# B&R Automation Studio project TD52 (part 7)

#### GeACtr.st
```iecst
(********************************************************************
 * COPYRIGHT -- INNIO Company
 ********************************************************************
 * Package:
 * File: GeACtr.st
 * Author: maierm
 * Created: May 22, 2012
 *******************************************************************)

(* ******************************************************************
 * History:
 *
 * V0.10.0		22-05-2012 maierm, 	generated
 * V0.10.1		21-06-2012 maierm, 	set clamp at line 102
 *								  	tProcPar.valid commented
 *								   	line 321 simplified - if / else
 *									was not necessary
 * V0.20.0		22-04-2013 maierm,	Datatype tParameter.Kp_manualAdjust, tParameter.Tn_manualAdjust and tParameter.Tv_manualAdjust
 *									changed to REAL, scaling included:
 *										tInput.Y_man 				==> tInput.Y_man * SCALE_PERCENT
 *										tInput.Y_set 				==> tInput.Y_set * SCALE_PERCENT
 *										tInput.A	 				==> tInput.A * SCALE_PERCENT
 *										tOutput.Y	 				==> rY / SCALE_PERCENT
 *										tOutput.e	 				==> xLCRPID.e / SCALE_PERCENT
 *										tOutput.Tn_tune 			==> tProcPar.Tn_tune * SCALE_TIME
 *										tOutput.Tv_tune 			==> tProcPar.Tv_tune * SCALE_TIME
 *										tParameter.Y_min   			==> tParameter.Y_min * SCALE_PERCENT
 *										tParameter.Y_max   			==> tParameter.Y_max * SCALE_PERCENT
 *										tParameter.dY_max  			==> tParameter.dY_max * SCALE_PERCENT
 *										tParameter.Y_block 			==> tParameter.Y_block * SCALE_PERCENT
 *										tParameter.Tn	   			==> tParameter.Tn / SCALE_TIME
 *										tParameter.Tv	   			==> tParameter.Tv / SCALE_TIME
 *										tParameter.Kp_manualAdjust 	==> tParameter.Kp_manualAdjust * SCALE_PERCENT
 *										tParameter.Tn_manualAdjust  ==> tParameter.Tn_manualAdjust * SCALE_PERCENT
 *										tParameter.Tv_manualAdjust 	==> tParameter.Tv_manualAdjust * SCALE_PERCENT
 *										tParameter.t_min_pulse_up 	==> tParameter.t_min_pulse_up / SCALE_TIME
 *										tParameter.t_period_up 		==> tParameter.t_period_up / SCALE_TIME
 *										tParameter.t_min_pulse_down ==> tParameter.t_min_pulse_down / SCALE_TIME
 *										tParameter.t_period_down 	==> tParameter.t_period_down / SCALE_TIME
 * V0.30.0		11-06-2013 maierm, 	comment format changed,
 *								   	corrected bug in part "input pwm up" and "input pwm down" -
 *								   	instead of bSafe2 was bSafe1 written - correct is bSafe2,
 *								   	changed rYmin to tParameter.Y_min in part "reset tuning or pid error",
 *								   	changed rYmax to tParameter.Y_max in part "reset tuning or pid error",
 *								   	set X to W for one cycle at enable of the fub
 * V0.40.0		27-06-2013 maierm, 	status of LCRPWM_up and LCRPWM_down has the lowest priority,
 *								   	instead of manuel mode, Input.Y_man is always following Output.Y,
 *								   	setting the internal I - component of the LCRPIDTune FUB directly to the new Y_min and Y_max limits
 * V0.50.0		28.06.2013 maierm, 	tInput.enable = FALSE sets the LCRPID to manual mode. LCRPID and LCRPIDTune is always running
 * V0.60.0		03.07.2013 Tinello,	Change tOutput.e  ==> Difference between W and X
 * V0.60.1		03.09.2013 maierm, 	bug at the feature "setting the internal I - component of the LCRPIDTune..." removed (Comparison
 *								   	between scaled and not scaled value)
 * V0.60.2		02.12.2013 Tinello,	If Y_Min = Y_Max -> automatic adjustment of Y_Min and Y_Max
 *									automatic limitation of Y_Min and Y_Max to -100% to 100%
 * V0.60.3		24.09.2016 Fahring,	set tAddPar.Kfbk = 1.0 to activate anti wind up protection
									set tAddPar.Tf_Tv = 0.1 / default value
 * V0.60.4		11.01.2017 Tinello,	Setpoint ramp changed from stage per second to linear ramp according to used cycle time
 * V0.70.0		25.01.2022 Perktold,Parameters: added W_set2, and GeinScheduling PID values; deleted "_manualAdjust" Parameters
									added Inputs: 	W_set2_Active, Retrigger, GainScheduling, Y_min_cust, Y_max_cust, AlwaysUseYRamp, KeepYManAtBlock
									added Outputs: 	Y_min_act, Y_max_act, Kp_act, Tn_act, Tv_act, Yp, Yi, Yd, BlockAutoTune, Show_PID_act
									LCRPWM replaced by LCRContinServo for sept_up/down output computation
 ****************************************************************************************************************************************************)

FUNCTION_BLOCK GeACtr

	(* ******************************** *)
	(*				ACCESS				*)
	(* ******************************** *)

	tParameter ACCESS pParameter; 								(* parameter from user *)
	tInput 	   ACCESS pInput;	  								(* input from user *)
	tOutput    ACCESS pOutput;	 								(* output from user *)
	tProcPar   ACCESS ADR(xLCRPIDTune.processPar);				(* Kp, Tn, Tv from LCRPIDTune *)

	(* ************************************************ *)
	(*	enable / auto / man / safe1 / safe2 / Retrigger	*)
	(* ************************************************ *)

	xR_TRIG_enable(CLK := tInput.enable);						(* generate rising trigger at enable*)
	bAuto  := tInput.enable AND NOT(tInput.Y_man_Active);		(* automatic *)
	bMan   := tInput.enable AND tInput.Y_man_Active;			(* manual *)
	bSafe1 := NOT(tInput.enable) AND NOT(tInput.Y_set_Active);	(* 1st safe - Y_block *)
	bSafe2 := NOT(tInput.enable) AND tInput.Y_set_Active;		(* 2nd safe - Y_set *)
	xR_TRIG_Retrigger(CLK := tInput.Retrigger);					(* generate rising trigger at retrigger*)

	(* ******************************** *)
	(*				  W					*)
	(* ******************************** *)

	tParameter.W_set := LIMIT(tParameter.W_min, tParameter.W_set, tParameter.W_max);	(* limit W from visu *)
	tParameter.W_set2 := LIMIT(tParameter.W_min, tParameter.W_set2, tParameter.W_max);	(* limit W from visu *)

	IF tInput.W_ext_Active 	THEN rWSet := tInput.W_ext; 					(* W from external *)
						 	ELSE
								IF tInput.W_set2_Active THEN
									rWSet := tParameter.W_set2;				(* W from visu - second internal set point*)
								ELSE
									rWSet := tParameter.W_set;				(* W from visu *)
								END_IF
							END_IF

	xLCRRamp_WSet.enable 	:= TRUE;
	xLCRRamp_WSet.dy_up 	:= tParameter.dW_up;							(* ramp up:   value/s *)
	xLCRRamp_WSet.dy_down 	:= tParameter.dW_down;							(* ramp down: value/s *)
	xLCRRamp_WSet.y_min 	:= tParameter.W_min;							(* limit W actual *)
	xLCRRamp_WSet.y_max 	:= tParameter.W_max;							(* limit W actual *)
	xLCRRamp_WSet.y_set 	:= tInput.X;									(* set X to W at enable of fub or retriggering *)
	xLCRRamp_WSet.set 		:= xR_TRIG_enable.Q OR xR_TRIG_Retrigger.Q;		(* activate set in case of retriggering or at enable of fub *)
	xLCRRamp_WSet(x 		:= rWSet);

	rW := LIMIT(tParameter.W_min, xLCRRamp_WSet.y, tParameter.W_max);		(* limit W *)
	tOutput.W 	:= rW; 														(* W actual *)

	(* ******************************** *)
	(*	 Y_min / Y_max (error 12037)	*)
	(* ******************************** *)

	IF (tParameter.Y_min <> rYMinOld) AND (tParameter.Y_min > tParameter.Y_max) THEN		(* Limit Y_min parameter to Y_max if Y_min > Y_max*)
		tParameter.Y_min := tParameter.Y_max;
	END_IF
	IF (tParameter.Y_max <> rYMaxOld) AND (tParameter.Y_max < tParameter.Y_min) THEN		(* Limit Y_max parameter to Y_min if Y_max < Y_min*)
		tParameter.Y_max := tParameter.Y_min;
	END_IF

	IF (tParameter.Y_max > Y_MAX  			OR												(* create error 12037 manually because of a bug in V2.80.1 *)
		tParameter.Y_min < Y_MIN 			OR
		tParameter.Y_max < tParameter.Y_min)
	THEN
		rYMax := 0;	 																		(* set Ymax to 0 *)
		rYMin := 0;  																		(* set Ymin to 0 *)
	ELSE
		rYMax := LIMIT(-1.0, MAX(MIN(tParameter.Y_max, tInput.Y_max_cust), MAX(tParameter.Y_min, tInput.Y_min_cust)), 1.0) * SCALE_PERCENT;	(* include Y_min_cust & Y_max_cust *)
		rYMin := LIMIT(-1.0, MIN(MAX(tParameter.Y_min, tInput.Y_min_cust), MIN(tParameter.Y_max, tInput.Y_max_cust)), 1.0) * SCALE_PERCENT;	(* include Y_min_cust & Y_max_cust *)
	END_IF

	IF rYMax = rYMin THEN																	(* in case Ymax = Ymin set them 0.01 appart *)
		IF rYMax >= 0 THEN	rYMin := rYMax - 0.01; 	END_IF
		IF rYMax < 0 THEN	rYMax := rYMin + 0.01; 	END_IF
	END_IF

	(* put the resulting YMin & YMax to the output structure *)
	tOutput.Y_max_act	:=	rYMax / SCALE_PERCENT;
	tOutput.Y_min_act	:=	rYMin / SCALE_PERCENT;

	(* If Y_min or Y_max is changed, the internal I - component of the LCRPIDTune FUB ran through the whole range to the new Y_min and
	(* Y_max limits. This behavior is optimised by setting the internal I - component of the LCRPIDTune FUB directly to the new Y_min and
	(* Y_max limits *)
	IF (rYMin <> rYMinintOld OR rYMax <> rYMaxintOld) THEN
		pYi1 ACCESS ADR(xLCRPIDTune.internal_data.Yi1); 									(* internal I - component can't be changed directly *)

		IF 	  (tOutput.Y <= (rYMin / SCALE_PERCENT)) THEN	pYi1 := rYMin;					(* set the internal I - component directly *)
		ELSIF (tOutput.Y >= (rYMax / SCALE_PERCENT)) THEN	pYi1 := rYMax;	END_IF			(* set the internal I - component directly *)
	END_IF

	IF xR_TRIG_Retrigger.Q OR xR_TRIG_enable.Q THEN											(* in case of retriggering or at enable of fub     *)
		pYi1 ACCESS ADR(xLCRPIDTune.internal_data.Yi1); 									(* access the internal integrator value of the CTR *)
		pYi1 := tOutput.Y * SCALE_PERCENT;													(* set the integrator to represent the last Y      *)
	END_IF;

	(* ******************************** *)
	(*				Tuning				*)
	(* ******************************** *)

	(* limit gain scheduling input from 0 to 1*)
	tInput.GainScheduling	:= LIMIT(0.0, tInput.GainScheduling, 1.0);

	(* Generate Output for VISU to decide if Parameters or actual PID-values are shown *)
	IF (tInput.GainScheduling >= 0.01) THEN
		tOutput.Show_PID_act	:= TRUE;		(* not show PID-paramters - show actual PID-values instead *)
	ELSE
		tOutput.Show_PID_act	:= FALSE;		(* show PID-paramters *)
	END_IF;

	(* De-/Activation of the Auto Tune function *)
	IF 	(xLCRPIDTune.status = 65534) 	OR		(* Auto Tune inactive (eg. Controller not enabled) *)
		(tInput.GainScheduling >= 0.01)	OR 		(* Gain Scheduling active - don't show parameters - show actual values instead *)
		NOT tInput.enable				OR		(* Controller nor enabled *)
		bMan									(* Controller running in manual mode *)
	THEN
		tInput.Tune_start 		:= FALSE;		(* reset *)
		tOutput.BlockAutoTune	:= TRUE;		(* lock VISU Button for AUTO Tune *)
	ELSE
		tOutput.BlockAutoTune	:= FALSE;		(* unlock VISU Button for AUTO Tune *)
	END_IF;

	(* tuning enable *)
	bTune_enable := TRUE;

	(* start *)
	IF (tInput.Tune_start = TRUE AND bAuto = TRUE AND usTune_status = 0) THEN (* user start *)
		bTune_active        := TRUE; 					(* tuning started *)
		bTunePIOld			:= tInput.Tune_PI;  		(* store *)
		bTunePIDOld			:= tInput.Tune_PID; 		(* store *)
		xLCRPIDTune.request := xTunReq(tInput.Tune_PI, tInput.Tune_PID, tInput.Tune_quality, tParameter.invert); (* calculate tuning request *)
	END_IF
	tInput.Tune_start 		:= FALSE;	(* reset *)

	(* stop *)
	IF (tInput.Tune_stop = TRUE 										OR 		(* user stop *)
		EDGENEG(bAuto) = TRUE											OR  	(* fub enable = FALSE OR manual = TRUE *)
		tAddPar.invert <> tParameter.invert 							OR  	(* invert parameter changed *)
		(xLCRPIDTune.status >= 12025 AND xLCRPIDTune.status <> 65534)) 			(* error happened *)
	THEN
		xLCRPIDTune.request := LCRPID_TUNE_REQU_OFF; 							(* deactivate tuning *)
		usTune_status       := 0; 												(* reset *)
		bTune_save 		    := FALSE; 											(* tuning stopped *)
		bTune_active        := FALSE; 											(* tuning stopped *)

		IF (xLCRPIDTune.status >= 12025 AND xLCRPIDTune.status <> 65534) THEN	(* tuning error *)
			usTune_status := xLCRPIDTune.status;								(* error status *)
			IF (xLCRPIDTune.status = 12039)	THEN
				usTune_status := xLCRPIDTune.addInfo;							(* show additional info *)
			ELSIF (xLCRPIDTune.status = 31564) THEN
				xResErr(ADR(bTune_enable), xLCRPIDTune.status);					(* reset enable after error *)
			END_IF
		END_IF
	END_IF
	tInput.Tune_stop := FALSE;			(* reset *)

	(* store tuning parameter *)
	IF (tInput.Tune_takeover = TRUE) THEN 						(* get tuning parameter every time *)
		bTune_save 	  		:= FALSE; 							(* tuning save closed *)
		usTune_status 		:= 0;	    						(* set status - no error / tuning finished / parameter saved *)
		tParameter.Kp 		:= tOutput.Kp_tune;
		tParameter.Tn 		:= tOutput.Tn_tune;
		tParameter.Tv 		:= tOutput.Tv_tune;
	END_IF
	tInput.Tune_takeover	:= FALSE; 	(* reset *)

	(* set ctrl parameter *)
	IF (bTune_active = FALSE AND bTune_save = TRUE) THEN 		(* no tuning / tuning parameter not set *)
		IF (bTunePIOld = TRUE AND bTunePIDOld = FALSE) THEN 	(* PI - tuning *)
			tProcPar.Tv_tune := 0;		(* delete D *)
		ELSIF (bTunePIOld = FALSE AND bTunePIDOld = FALSE) THEN (* P - tuning *)
			tProcPar.Tn_tune := 0;		(* delete I *)
			tProcPar.Tv_tune := 0;		(* delete D *)
		END_IF
		tOutput.Kp_tune := tProcPar.Kp_tune; 			  		(* fub to tune parameter *)
		tOutput.Tn_tune := tProcPar.Tn_tune * SCALE_TIME; 		(* fub to tune parameter *)
		tOutput.Tv_tune := tProcPar.Tv_tune * SCALE_TIME; 		(* fub to tune parameter *)

	ELSIF (bTune_active = FALSE AND bTune_save = FALSE) THEN 	(* no tuning and parameter set *)
		tProcPar.valid   := TRUE; 										(* necessary for the LCRPIDTune(). Kp_tune, Tn_tune and Tv_tune *)
																		(* are "valid" and can be used from the FUB 					*)
		(* Interpolate PID-Parameters via Gain Scheduling *)
		tProcPar.Kp_tune :=  (1.0 - tInput.GainScheduling) * tParameter.Kp + tInput.GainScheduling * tParameter.Kp_GainScheduling; 						(* parameter to fub *)
		tProcPar.Tn_tune := ((1.0 - tInput.GainScheduling) * tParameter.Tn + tInput.GainScheduling * tParameter.Tn_GainScheduling) / SCALE_TIME; 		(* parameter to fub *)
		tProcPar.Tv_tune := ((1.0 - tInput.GainScheduling) * tParameter.Tv + tInput.GainScheduling * tParameter.Tv_GainScheduling) / SCALE_TIME; 	 	(* parameter to fub *)
		IF xR_TRIG_Retrigger.Q OR xR_TRIG_enable.Q THEN
			tProcPar.Tv_tune := 0;
		END_IF;
	END_IF

	(* tuning status *)
	IF (bTune_active = FALSE AND bTune_save = TRUE) THEN
		usTune_status := 1; 									(* set status - tuning finished, but not closed *)
	ELSIF (bTune_active = TRUE) THEN
		usTune_status := 2;										(* set status - tuning active *)
	END_IF

	(* parameter *)
	xLCRPIDTune.enable 			:= bTune_enable;
	xLCRPIDTune.Y_min  			:= rYMin;
	xLCRPIDTune.Y_max  			:= rYMax;
	xLCRPIDTune.X_min  			:= tInput.X_min;
	xLCRPIDTune.X_max  			:= tInput.X_max;
	xLCRPIDTune.P_manualAdjust 	:= 0;
	xLCRPIDTune.I_manualAdjust 	:= 0;
	xLCRPIDTune.D_manualAdjust 	:= 0;

	(* additional parameter *)
	tAddPar.dY_max      		:= tParameter.dY_max * SCALE_PERCENT;
	tAddPar.deadband    		:= tParameter.deadband;
	tAddPar.d_mode      		:= LCRPID_D_MODE_E;
	tAddPar.invert	    		:= tParameter.invert;
	tAddPar.Kfbk				:= 1.0;
	tAddPar.Tf_Tv				:= 0.1;
	xLCRPIDTune.pAddPar 		:= ADR(tAddPar);	 (* additional parameter *)

	(* reset valid *)
	IF (EDGEPOS(bTune_active) = TRUE) THEN 	(* new tuning *)
		tProcPar.valid 			:= FALSE;  	(* reset necessary at new tuning - otherwise ctrl fub is immediately finished *)
	END_IF

	xLCRPIDTune();

	(* put the resulting PID-values to the output structure *)
	tOutput.Kp_act	:= tProcPar.Kp_tune;
	tOutput.Tn_act	:= tProcPar.Tn_tune * SCALE_TIME;
	tOutput.Tv_act	:= tProcPar.Tv_tune * SCALE_TIME;

	(* store during tuning the parameters from the visu to the internal structure (if user changed it during the tuning) *)
	IF (bTune_active = TRUE AND xLCRPIDTune.state < LCRPID_TUNE_STATE_RESET_CNTL) THEN
		tProcPar.Kp_tune 	  := tParameter.Kp; 			 (* parameter to fub *)
		tProcPar.Tn_tune 	  := tParameter.Tn / SCALE_TIME; (* parameter to fub *)
		tProcPar.Tv_tune 	  := tParameter.Tv / SCALE_TIME; (* parameter to fub *)
	END_IF

	(* set parameter after enable = TRUE (LCRPID sets parameter to 0 / 0.5 aso. after enable = TRUE) *)
	IF (EDGEPOS(tInput.enable) = TRUE) THEN
		tProcPar.valid   	  := TRUE; 		   				 (* valid necessary that controller use the parameters - after enable = TRUE *)
		tProcPar.Kp_tune 	  := tParameter.Kp; 			 (* parameter to fub *)
		tProcPar.Tn_tune 	  := tParameter.Tn / SCALE_TIME; (* parameter to fub *)
		tProcPar.Tv_tune 	  := tParameter.Tv / SCALE_TIME; (* parameter to fub *)
	END_IF

	(* tuning finished *)
	IF (bTune_active = TRUE AND xLCRPIDTune.state = LCRPID_TUNE_STATE_FINISHED) THEN
		xLCRPIDTune.request   := LCRPID_TUNE_REQU_OFF; 		(* deactivate tuning *)
		bTune_save 		      := TRUE;  					(* save parameter *)
		bTune_active          := FALSE; 					(* tuning finished *)

		(* error 12041 manually *)
		IF (tProcPar.valid = FALSE AND rW <> rWOld) THEN	(* set status 12041 manually because of a bug in V2.80.1 *)
			rWOld 		      := rW;
			bTune_save        := FALSE;
			usTune_status     := 12041;
		END_IF
	END_IF

	(* error 12041 manually *)
	IF (bTune_active = FALSE) THEN
		rWOld := rW;
	END_IF

	(* ******************************** *)
	(*				PID					*)
	(* ******************************** *)

	(* error *)
	IF (xLCRPID.status >= 12025 AND xLCRPID.status <> 65534) THEN	 (* error happened *)
		usPID_status := xLCRPID.status;	 			(* show error number *)
	ELSE
		usPID_status := 0;
	END_IF

	(* Y manual *)
	IF (bSafe1 = TRUE) THEN											(* first safe value *)
		IF tInput.KeepYManAtBlock THEN								(* prevent overriding of tInput.Y_man *)
			xLCRPID.Y_man:= tParameter.Y_block * SCALE_PERCENT;		(* write Y_block value to LCRPID directly *)
		ELSE
			tInput.Y_man := tParameter.Y_block;						(* override Y_man with Y_block value*)
		END_IF;
		xLCRPID.mode := LCRPID_MODE_MAN_JOLTFREE;					(* PID manual mode *)
	END_IF

	IF (bSafe2 = TRUE) THEN 										(* second safe value *)
		IF tInput.KeepYManAtBlock THEN								(* prevent overriding of tInput.Y_man *)
			xLCRPID.Y_man:= tInput.Y_set * SCALE_PERCENT;			(* write Y_set value to LCRPID directly *)
		ELSE
			tInput.Y_man := tInput.Y_set;							(* override Y_man with Y_set value*)
		END_IF
		xLCRPID.mode := LCRPID_MODE_MAN_JOLTFREE;					(* PID manual mode *)
	END_IF

	IF (bAuto = TRUE) THEN											(* automatic mode *)
		tInput.Y_man := tOutput.Y;									(* in automatic mode Y_man is following Y *)
		xLCRPID.Y_man:= tInput.Y_man * SCALE_PERCENT;				(* write Y_man value to LCRPID directly *)
		xLCRPID.mode := LCRPID_MODE_AUTO;							(* PID automatic mode *)
	END_IF

	IF (bMan = TRUE) THEN																	(* manual mode *)
		tInput.Y_man := LIMIT(rYMin / SCALE_PERCENT, tInput.Y_man, rYMax / SCALE_PERCENT);	(* limit Y manual from visu *)
		xLCRPID.Y_man := tInput.Y_man * SCALE_PERCENT;										//Y_man for LCRPID acc Y_man
		xLCRPID.mode := LCRPID_MODE_MAN_JOLTFREE;											(* PID manual mode *)
	END_IF

	IF NOT tInput.KeepYManAtBlock THEN
		xLCRPID.Y_man 	 := tInput.Y_man * SCALE_PERCENT;									(* transfer Y_man value to LCRPID *)
	END_IF;

	(* parameter *)
	xLCRPID.enable 	 := TRUE;
	xLCRPID.ident  	 := xLCRPIDTune.ident;
	xLCRPID.Y_max  	 := rYMax;
	xLCRPID.Y_min  	 := rYMin;
	xLCRPID.A	   	 := tInput.A * SCALE_PERCENT;
	xLCRPID.W 		 := rW;		   					(* W *)
	xLCRPID.X 		 := tInput.X;  					(* X *)
	xLCRPID();

	rY 		  		 := xLCRPID.Y;					(* Y FuB *)
	tOutput.e 		 := xLCRPID.X - xLCRPID.W;		(* Error = X - W *)

	(* ******************************** *)
	(*				  Y 				*)
	(* ******************************** *)

	(* change of request *)
	IF ((EDGEPOS(bTune_active) = TRUE) OR 							(* set Y to Y old after start of tuning *)
		(EDGENEG(bTune_active) = TRUE AND bTune_save = FALSE)) 		(* set Y to Y old after tuning stop 	*)
	THEN
		rY := rYOld;	(* Y decreases minimal for one cycle after start of tuning and cancel of tuning	*)
					   	(* - set Y to YOld for one cycle compensate this decrease 						*)
	END_IF
	rYOld := rY;

	(* first safe value *)
	IF (bSafe1 = TRUE) THEN
		rY := tParameter.Y_block * SCALE_PERCENT;	(* Y_block *)
	END_IF

	(* second safe value *)
	IF (bSafe2 = TRUE) THEN
		rY := tInput.Y_set * SCALE_PERCENT;			(* Y_set *)
	END_IF

	(* additional ramp at the end of the controller to prohibit step changes on Y *)
	xLCRRamp_Y.enable 	:= TRUE;
	xLCRRamp_Y.dy_up 	:= tParameter.dY_max;			(* ramp up:   value/s *)
	xLCRRamp_Y.dy_down 	:= tParameter.dY_max;			(* ramp down: value/s *)
	xLCRRamp_Y.y_min 	:= -1.0;						(* limit Y actual - full range *)
	xLCRRamp_Y.y_max 	:=  1.0;						(* limit Y actual - full range *)
	xLCRRamp_Y.y_set 	:= rY / SCALE_PERCENT;
	xLCRRamp_Y.set 		:= NOT tInput.AlwaysUseYRamp;	(* possibility to deactivate the ramp *)
	xLCRRamp_Y(x 		:= (rY / SCALE_PERCENT));

	tOutput.Y := xLCRRamp_Y.y; 				(* Y to output *)

	(* transfer all parts of Y to the tOutput structure *)
	tOutput.Yp		:= xLCRPID.Yp / SCALE_PERCENT;
	tOutput.Yi		:= xLCRPID.Yi / SCALE_PERCENT;
	tOutput.Yd		:= xLCRPID.Yd / SCALE_PERCENT;

	(* ******************************** *)
	(*				PWM					*)
	(* ******************************** *)
	IF tInput.StepperMode THEN
		(* PWM Up *)
		(* enable *)
		bPWM_up_enable := tInput.enable;		(* activate *)
		xResChg(ADR(bPWM_up_enable), tParameter.t_min_pulse_up / SCALE_TIME, xLCRPWM_up.t_min_pulse);		(* reset enable if t_min_pulse
																											   changed *)
		(* parameter *)
		xLCRPWM_up.enable 	   := bPWM_up_enable;
		xLCRPWM_up.max_value   := rYMax;
		xLCRPWM_up.min_value   := xCalMid(rYMin, rYMax);		(* calculate middle of Y_max / Y_min range *)
		xLCRPWM_up.t_min_pulse := tParameter.t_min_pulse_up / SCALE_TIME;
		xLCRPWM_up.t_period	   := tParameter.t_period_up / SCALE_TIME;

		(* input PWM Up *)
		IF (bSafe1 = TRUE OR bSafe2 = TRUE OR bMan = TRUE) 		(* Y_block / Y_set / Y_man *)
		THEN
			xLCRPWM_up.x := xCalMid(rYMin, rYMax); 				(* restrict input to middle of Y_max / Y_min range *)
		ELSE
			xLCRPWM_up.x := rY; 								(* actual value *)
		END_IF

		xLCRPWM_up();

		(* PWM Down *)
		(* enable *)
		bPWM_down_enable := tInput.enable;		(* activate *)
		xResChg(ADR(bPWM_down_enable), tParameter.t_min_pulse_down / SCALE_TIME, xLCRPWM_down.t_min_pulse);	(* reset enable if t_min_pulse
																											   changed *)
		(* parameter *)
		xLCRPWM_down.enable 	 := bPWM_down_enable;
		xLCRPWM_down.max_value   := xCalMid(rYMin, rYMax);		(* calculate middle of Y_max / Y_min range *)
		xLCRPWM_down.min_value   := rYMin;
		xLCRPWM_down.t_min_pulse := tParameter.t_min_pulse_down / SCALE_TIME;
		xLCRPWM_down.t_period	 := tParameter.t_period_down / SCALE_TIME;

		(* input PWM Down *)
		IF (bSafe1 = TRUE OR bSafe2 = TRUE OR bMan = TRUE) 		(* Y_block / Y_set / Y_man *)
		THEN
			xLCRPWM_down.x := xCalMid(rYMin, rYMax); 			(* restrict input to middle of Y_max / Y_min range *)
		ELSE
			xLCRPWM_down.x := rY;								(* actual value *)
		END_IF

		xLCRPWM_down();

		(* PWM Up / PWM Down *)
		(* common status for PWM Up and PWM Down *)
		IF 	  (xLCRPWM_up.status   >= 12025) THEN	usPWM_status := xLCRPWM_up.status;
		ELSIF (xLCRPWM_down.status >= 12025) THEN	usPWM_status := xLCRPWM_down.status;
											 ELSE	usPWM_status := 0;				 		END_IF

		(* output only if PWM Up and PWM Down has no error *)
		IF (usPWM_status = 0) THEN
			tOutput.Step_up   := xLCRPWM_up.pulse;
			tOutput.Step_down := NOT(xLCRPWM_down.pulse); 	(* invert necessary *)
		ELSE
			tOutput.Step_up   := FALSE;
			tOutput.Step_down := FALSE;
		END_IF

	ELSE  // tInput.StepperMode = FALSE

		(* ******************************** *)
		(*     continuous servo drive   	*)
		(* ******************************** *)

		(* Enable servo drive *)
		xLCRContinServo.enable        := tInput.enable;

		(* Parameters for continuous servo drive *)
		xLCRContinServo.max_value     := tOutput.Y_max_act;
		xLCRContinServo.min_value     := tOutput.Y_min_act;
		xLCRContinServo.t_impulse     := (tParameter.t_min_pulse_up / 1000) ;
		IF tParameter.dY_max <> 0 THEN
			xLCRContinServo.t_change_up   := (1 / tParameter.dY_max) * (tOutput.Y_max_act - tOutput.Y_min_act);
			xLCRContinServo.t_change_down := (1 / tParameter.dY_max) * (tOutput.Y_max_act - tOutput.Y_min_act);
		END_IF;

		(* Continuous servo drive *)
		xLCRContinServo.x   := tOutput.Y;
		xLCRContinServo();										(* LCRContinServo function block call *)

		(* Copy up and down to controller output *)
		tOutput.Step_up 		:= xLCRContinServo.up;
		tOutput.Step_down 		:= xLCRContinServo.down;
	END_IF;

	(* ******************************** *)
	(*		reset status LCRPIDTune		*)
	(* ******************************** *)

	(* reset tuning or pid error *)
	IF (tParameter.Kp   			<> rKpOld  				OR
		tParameter.Tn 	 			<> rTnOld  				OR
		tParameter.Tv   			<> rTvOld  				OR
		tParameter.Y_min 			<> rYMinOld 			OR
		tParameter.Y_max 			<> rYMaxOld 			OR
		rYMinintOld					<> rYMin				OR
		rYMaxintOld					<> rYMax				OR
		tInput.X_min     			<> rXMinOld 			OR
		tInput.X_max     			<> rXMaxOld 			OR
		tParameter.deadband 		<> rDeadbandOld			OR
		tParameter.dY_max			<> rDYMaxOld)
	THEN
		IF (usTune_status >= 12025 AND usTune_status <> 65534) THEN
			usTune_status := 0;	(* reset tune status after error *)
		END_IF
	END_IF

	rKpOld   			:= tParameter.Kp; (* restore *)
	rTnOld   			:= tParameter.Tn;
	rTvOld   			:= tParameter.Tv;
	rYMinOld 			:= tParameter.Y_min;
	rYMaxOld 			:= tParameter.Y_max;
	rYMinintOld			:= rYMin;
	rYMaxintOld			:= rYMax;
	rXMinOld 			:= tInput.X_min;
	rXMaxOld 			:= tInput.X_max;
	rDeadbandOld      	:= tParameter.deadband;
	rDYMaxOld		  	:= tParameter.dY_max;

	(* ******************************** *)
	(*				Status				*)
	(* ******************************** *)

	tOutput.Active := tInput.enable;

	IF (tInput.enable = TRUE) THEN	(* fub enable *)

		IF 	  (xChkStat(usPID_status)  = TRUE) THEN	tOutput.status := usPID_status;		(* LCRPID state *)
		ELSIF (xChkStat(usTune_status) = TRUE) THEN tOutput.status := usTune_status;	(* LCRTune state *)
		ELSIF (xChkStat(usPWM_status)  = TRUE) THEN tOutput.status := usPWM_status; 	(* LCRPWM_up AND LCRPWM_down state *)
											   ELSE tOutput.status := 0;
		END_IF

	ELSE							(* fub disable *)
		usTune_status  := 0;		(* reset *)
		usPID_status   := 0;
		usPWM_status   := 0;
		bTune_active   := FALSE;
		bTune_save     := FALSE;
		tOutput.status := 65534;	(* status enable = FALSE *)
	END_IF

END_FUNCTION_BLOCK
```

#### GeACtrFunc.st - Functions of the library
```iecst
(********************************************************************
 * COPYRIGHT -- INNIO Company
 ********************************************************************
 * Package:
 * File: GeACtrFunc.st
 * Author: maierm
 * Created: May 22, 2012
 *******************************************************************)

(* ******************************************************************
 * History:
 *
 * V0.1.0		22-05-2012	maierm, generated
 *
 *
 *
 *******************************************************************)

(* returns the middle of min and max value *)
FUNCTION xCalMid

	xCalMid := rMin + (rMax - rMin) / 2;

END_FUNCTION

(* returns TRUE if status is between 0 and 65534  *)
FUNCTION xChkStat

	IF (usActStatus <> 0 AND usActStatus <> 65534) THEN
		xChkStat := TRUE;
	ELSE
		xChkStat := FALSE;
	END_IF

END_FUNCTION

(* switch off the enable if parameter changed *)
FUNCTION xResChg

	bEnable ACCESS pEnable;

	IF (rAct <> rOld) THEN	(* check if old value is different to actual value *)
		bEnable := FALSE;	(* reset *)
	END_IF

	xResChg;

END_FUNCTION

(* reset the enable if an error happened *)
FUNCTION xResErr

	bEnable ACCESS pEnable;

	IF (usStatus >= 12025 AND usStatus <> 65534) THEN	(* switch off enable *)
		bEnable := FALSE;
	END_IF

	xResErr;

END_FUNCTION

(* returns the tuning request *)
FUNCTION xTunReq

	xTunReq := 0;
	xTunReq := xTunReq + LCRPID_TUNE_REQU_OSCILLATE;	(* oscillation *)

	IF (bInvert = TRUE) THEN
		xTunReq := xTunReq + LCRPID_TUNE_REQU_DIR_NEG;		(* negative direction *)
	ELSE
		xTunReq := xTunReq + LCRPID_TUNE_REQU_DIR_POS;		(* positive direction *)
	END_IF

	IF (bPI = TRUE) THEN
		IF (bPID = TRUE) THEN	(* PID tuning *)
			xTunReq := xTunReq + LCRPID_TUNE_REQU_PID;
		ELSE					(* PI tuning *)
			xTunReq := xTunReq + LCRPID_TUNE_REQU_PI;
		END_IF
	ELSE						(* P tuning *)
		xTunReq := xTunReq + LCRPID_TUNE_REQU_P;
	END_IF

	IF (ssQuality = 0) THEN		(* 1 try - 3 periods *)
		xTunReq := xTunReq + LCRPID_TUNE_REQU_OSC_1 + LCRPID_TUNE_REQU_PER_3;
	ELSIF (ssQuality = 1) THEN	(* 2 tries - 4 periods *)
		xTunReq := xTunReq + LCRPID_TUNE_REQU_OSC_2 + LCRPID_TUNE_REQU_PER_4;
	ELSIF (ssQuality = 2) THEN	(* 3 tries - 5 periods *)
		xTunReq := xTunReq + LCRPID_TUNE_REQU_OSC_3 + LCRPID_TUNE_REQU_PER_5;
	END_IF

END_FUNCTION
```

### Library Logical/Libraries/CTRL (ANSIC, version 1.00.0)

#### CTRL.fun
```iecst
FUNCTION_BLOCK DigFil
	VAR_INPUT
		Input	:REAL;
		Ordnung	:UINT;
		an	:ARRAY[0..3] OF REAL;
		bn	:ARRAY[0..3] OF REAL;
	END_VAR
	VAR_OUTPUT
		Output	:REAL;
	END_VAR
	VAR
		Y	:ARRAY[0..3] OF REAL;
		X	:ARRAY[0..3] OF REAL;
	END_VAR
END_FUNCTION_BLOCK
```

#### digfilscr.c
```c
/***********************************************************************************
* Name      : digfilsrc.c
* Titel     : Regelungstechnik
* Version   : V0.1
* Datum     : 28.06.2006
*
* Uebergabe : Input		REAL	Eingangssignal
*			  Ordnung	USINT	Filterordnung
*			  an		REAL	Nennerkoeffizienten
*			  bn		REAL	Zählerkoeffizienten
*			  Output	REAL	Ausgangssignal
*			  Y			REAL	Zähler
*			  X			REAL	Nenner
*
*
* History   :
* V0.1		  28.06.2006,Hirzinger	erstellt
*
***********************************************************************************/
#include <CTRL.h>

unsigned int	uszaehl;
float			rN_N;

void DigFil(DigFil_typ *tDigFilVar)
{

	/***** EINGANG ********/
	/*tDigFilVar->X[3]	= tDigFilVar->X[2];
	tDigFilVar->X[2]	= tDigFilVar->X[1];
	tDigFilVar->X[1]	= tDigFilVar->X[0];
	tDigFilVar->X[0]	= tDigFilVar->Input;
	*/

	/***** HISTORIE EINGANG *****/
	for(uszaehl = tDigFilVar->Ordnung; uszaehl >= 1; uszaehl--)
		tDigFilVar->X[uszaehl] = tDigFilVar->X[uszaehl-1];

	tDigFilVar->X[0]	= tDigFilVar->Input;

	/********  ZÄHLER B*X **********/
	/*for (uszaehl = 0; uszaehl <= tDigFilVar->Ordnung; uszaehl++)
		rN_N	= rN_N + tDigFilVar->X[uszaehl] * tDigFilVar->bn[uszaehl];

	*/
	tDigFilVar->Y[0] = 	tDigFilVar->X[0] * tDigFilVar->bn[0] + tDigFilVar->X[1] * tDigFilVar->bn[1] + tDigFilVar->X[2] * tDigFilVar->bn[2] ;

	/********  NENNER A*Y **********/
	/*for (uszaehl = 1; uszaehl <= tDigFilVar->Ordnung; uszaehl++)
		rN_N	= rN_N - tDigFilVar->Y[uszaehl] * tDigFilVar->an[uszaehl];
	*/

	tDigFilVar->Y[0] = tDigFilVar->Y[0] - tDigFilVar->Y[1] * tDigFilVar->an[1] - tDigFilVar->Y[2] * tDigFilVar->an[2];

	/*tDigFilVar->Y[3]	= tDigFilVar->Y[2];
	tDigFilVar->Y[2]	= tDigFilVar->Y[1];
	tDigFilVar->Y[1]	= tDigFilVar->Y[0];
	*/

	/***** HISTORIE AUSGANG Z-1 *****/
	for (uszaehl = tDigFilVar->Ordnung; uszaehl >= 1; uszaehl--)
		tDigFilVar->Y[uszaehl]	= tDigFilVar->Y[uszaehl-1];

/*	tDigFilVar->Y[1]	= rN_N;*/

	/***** AUSGANG *******/
	tDigFilVar->Output	= tDigFilVar->Y[0];
}
```

### Library Logical/Libraries/lSimPID4 (ANSIC, version 0.01.0)

#### lSimPID4.fun
```iecst
FUNCTION_BLOCK SimPID4
  VAR_INPUT
    ssMethodType: SINT;
  END_VAR  VAR_INPUT
        P : REAL; (*Proportional Gain*)
  END_VAR
  VAR_INPUT
        I : REAL; (*Integral Gain*)
  END_VAR
  VAR_INPUT
        wxmin : LREAL; (*Minimum Input*)
  END_VAR
  VAR_INPUT
        deadband : LREAL; (*Deadband*)
  END_VAR
  VAR_INPUT
        D : REAL; (*Differential Gain*)
  END_VAR
  VAR_INPUT
        N : REAL; (*Filter Coefficient*)
  END_VAR
  VAR_INPUT
        umax : REAL; (*Upper Output Saturation Level*)
  END_VAR
  VAR_INPUT
        umin : REAL; (*Lower Output Saturation Level*)
  END_VAR
  VAR_INPUT
        Kt : REAL; (*Tracking Gain*)
  END_VAR
  VAR_INPUT
        wxmax : LREAL; (*Maximum Input*)
  END_VAR
  VAR_INPUT
        mode : USINT; (*Mode*)
  END_VAR
  VAR_INPUT
        u_man : REAL; (*Manual Value*)
  END_VAR
  VAR_INPUT
        a : REAL; (*Feedforward Value*)
  END_VAR
  VAR_INPUT
        invert : BOOL := FALSE; (*Invert*)
  END_VAR
  VAR_INPUT
        w : REAL; (*Reference Value*)
  END_VAR
  VAR_INPUT
        x : REAL; (*Actual Value*)
  END_VAR
  VAR_INPUT
        reset : BOOL := FALSE; (*Reset*)
  END_VAR
  VAR_INPUT
        I0 : REAL; (*I Integrator Reset*)
  END_VAR
  VAR_INPUT
        D0 : REAL; (*D Integrator Reset (Filter)*)
  END_VAR
  VAR_OUTPUT
        u : REAL; (*Controller Output*)
  END_VAR
  VAR_OUTPUT
        up : REAL; (*Proportional Output*)
  END_VAR
  VAR_OUTPUT
        ui : REAL; (*Integral Output*)
  END_VAR
  VAR_OUTPUT
        ud : REAL; (*Differential Output*)
  END_VAR
  VAR_OUTPUT
        u_tr : REAL; (*Tracking Output*)
  END_VAR
  VAR_INPUT
        fbk_mode : USINT; (*Anti Windup Feedback Mode*)
  END_VAR
  VAR_INPUT
        u_fbk : REAL; (*External Anti Windup Feedback Value*)
  END_VAR
	VAR
		bur_SimPID4_DWork : D_Work_SimPID4;
	END_VAR
	VAR
		bur_SimPID4_B : BlockIO_SimPID4;
	END_VAR
END_FUNCTION_BLOCK
```

#### lSimPID4.typ
```iecst
 TYPE

END_TYPE
TYPE
	D_Work_SimPID4 : STRUCT

		Integrator_DSTATE : REAL;
		Filter_DSTATE : REAL;
		Integrator_IC_LOADING : USINT;
		Filter_IC_LOADING : USINT;
	END_STRUCT;

	 BlockIO_SimPID4 : STRUCT

		Input10 : REAL;
		Input6 : REAL;
		Input4 : REAL;
		Input : REAL;
		Gain : REAL;
		Input2 : REAL;
		Integrator : REAL;
		Input3 : REAL;
		FilterCoefficient : REAL;
		Saturation : REAL;
		Modeswitch : REAL;
		Input8 : REAL;
		Input9 : USINT;
		Input7 : USINT;
		Input5 : BOOL;
		Input1 : BOOL;
	END_STRUCT;

END_TYPE
```

#### SimPID4.h
```c
/********************************************************************
 * COPYRIGHT -- Bernecker + Rainer Industrie-Elektronik Ges.m.b.H.
 ********************************************************************
 * Program: SimPID4
 * File: SimPID4.h
 * Author: 106001702
 * Created: Wed Nov 09 12:46:00 2011
 ********************************************************************
 * Header for program SimPID4
 ********************************************************************
 * Generated with B&R Automation Studio Target for Simulink V4.2
 * (ERT based)
 ********************************************************************/

#ifndef RTW_HEADER_SimPID4_h_
#define RTW_HEADER_SimPID4_h_
#ifndef SimPID4_COMMON_INCLUDES_
# define SimPID4_COMMON_INCLUDES_
#include <math.h>
#include "rtwtypes.h"
#endif                                 /* SimPID4_COMMON_INCLUDES_ */

#include "SimPID4_types.h"
#include "lSimPID4.h"

/* Macros for accessing real-time model data structure */
#ifndef rtmGetErrorStatus
# define rtmGetErrorStatus(rtm)        ((void*) 0)
#endif

#ifndef rtmSetErrorStatus
# define rtmSetErrorStatus(rtm, val)   ((void) 0)
#endif

#ifndef rtmGetStopRequested
# define rtmGetStopRequested(rtm)      ((void*) 0)
#endif

#ifndef MIN
#define MIN(a,b)                       ((a) < (b) ? (a) : (b))
#endif

#ifndef MAX
#define MAX(a,b)                       ((a) > (b) ? (a) : (b))
#endif

/* Block signals (auto storage) */

/* Block states (auto storage) for system '<Root>' */

/* Block signals (auto storage) */
extern BlockIO_SimPID4 SimPID4_B;

/* Block states (auto storage) */
extern D_Work_SimPID4 SimPID4_DWork;

/* Model entry point functions */
extern void SimPID4_initialize(struct SimPID4* inst);
extern void SimPID4_step(struct SimPID4* inst);
extern void SimPID4_terminate(struct SimPID4* inst);

/*-
 * The generated code includes comments that allow you to trace directly
 * back to the appropriate location in the model.  The basic format
 * is <system>/block_name, where system is the system number (uniquely
 * assigned by Simulink) and block_name is the name of the block.
 *
 * Use the MATLAB hilite_system command to trace the generated code back
 * to the model.  For example,
 *
 * hilite_system('<S3>')    - opens system 3
 * hilite_system('<S3>/Kp') - opens and selects block Kp which resides in S3
 *
 * Here is the system hierarchy for this model
 *
 * '<Root>' : SimPID4
 * '<S1>'   : SimPID4/Model Info
 * '<S2>'   : SimPID4/PID Autocoding
 * '<S3>'   : SimPID4/PID Autocoding/PID
 * '<S4>'   : SimPID4/PID Autocoding/PID/Clamping circuit
 * '<S5>'   : SimPID4/PID Autocoding/PID/Clamping circuit/Compare To Constant
 */
#endif                                 /* RTW_HEADER_SimPID4_h_ */
```

#### SimPID4_private.h
```c
/********************************************************************
 * COPYRIGHT -- Bernecker + Rainer Industrie-Elektronik Ges.m.b.H.
 ********************************************************************
 * Program: SimPID4
 * File: SimPID4_private.h
 * Author: 106001702
 * Created: Wed Nov 09 12:46:00 2011
 ********************************************************************
 * Header for program SimPID4
 ********************************************************************
 * Generated with B&R Automation Studio Target for Simulink V4.2
 * (ERT based)
 ********************************************************************/

#ifndef RTW_HEADER_SimPID4_private_h_
#define RTW_HEADER_SimPID4_private_h_
#include "rtwtypes.h"
#include <bur/plctypes.h>
#ifndef __RTWTYPES_H__
#error This file requires rtwtypes.h to be included
#else
#ifdef TMWTYPES_PREVIOUSLY_INCLUDED
#error This file requires rtwtypes.h to be included before tmwtypes.h
#else

/* Check for inclusion of an incorrect version of rtwtypes.h */
#ifndef RTWTYPES_ID_C08S16I32L32N32F1
#error This code was generated with a different "rtwtypes.h" than the file included
#endif                                 /* RTWTYPES_ID_C08S16I32L32N32F1 */
#endif                                 /* TMWTYPES_PREVIOUSLY_INCLUDED */
#endif                                 /* __RTWTYPES_H__ */

#ifndef MIN
#define MIN(a,b)                       ((a) < (b) ? (a) : (b))
#endif

#ifndef MAX
#define MAX(a,b)                       ((a) > (b) ? (a) : (b))
#endif

/* Imported (extern) block parameters */
extern real_T deadband;                /* Variable: deadband
                                        * Referenced by: '<S2>/Deadband'
                                        */
extern real_T wxmax;                   /* Variable: wxmax
                                        * Referenced by: '<S2>/Scaling'
                                        */
extern real_T wxmin;                   /* Variable: wxmin
                                        * Referenced by: '<S2>/Scaling'
                                        */
extern real32_T D;                     /* Variable: D
                                        * Referenced by: '<S3>/Gain2'
                                        */
extern real32_T I;                     /* Variable: I
                                        * Referenced by: '<S3>/Gain1'
                                        */
extern real32_T Kt;                    /* Variable: Kt
                                        * Referenced by: '<S2>/Constant'
                                        */
extern real32_T N;                     /* Variable: N
                                        * Referenced by: '<S3>/Filter Coefficient'
                                        */
extern real32_T P;                     /* Variable: P
                                        * Referenced by: '<S3>/Gain'
                                        */
extern real32_T umax;                  /* Variable: umax
                                        * Referenced by: '<S3>/Saturation'
                                        */
extern real32_T umin;                  /* Variable: umin
                                        * Referenced by: '<S3>/Saturation'
                                        */

#endif                                 /* RTW_HEADER_SimPID4_private_h_ */
```

#### SimPID4_types.h
```c
/********************************************************************
 * COPYRIGHT -- Bernecker + Rainer Industrie-Elektronik Ges.m.b.H.
 ********************************************************************
 * Program: SimPID4
 * File: SimPID4_types.h
 * Author: 106001702
 * Created: Wed Nov 09 12:46:00 2011
 ********************************************************************
 * Header for program SimPID4
 ********************************************************************
 * Generated with B&R Automation Studio Target for Simulink V4.2
 * (ERT based)
 ********************************************************************/

#ifndef RTW_HEADER_SimPID4_types_h_
#define RTW_HEADER_SimPID4_types_h_
#ifndef MIN
#define MIN(a,b)                       ((a) < (b) ? (a) : (b))
#endif

#ifndef MAX
#define MAX(a,b)                       ((a) > (b) ? (a) : (b))
#endif
#endif                                 /* RTW_HEADER_SimPID4_types_h_ */
```

#### rtwtypes.h
```c
/********************************************************************
 * COPYRIGHT -- Bernecker + Rainer Industrie-Elektronik Ges.m.b.H.
 ********************************************************************
 * Program: SimPID4
 * File: rtwtypes.h
 * Author: 106001702
 * Created: Wed Nov 09 12:46:00 2011
 ********************************************************************
 * Header for program SimPID4
 ********************************************************************
 * Generated with B&R Automation Studio Target for Simulink V4.2
 * (ERT based)
 ********************************************************************/

#ifndef RTW_HEADER_rtwtypes_h_
#define RTW_HEADER_rtwtypes_h_
#ifndef __RTWTYPES_H__
#define __RTWTYPES_H__
#ifndef TRUE
# define TRUE                          (1U)
#endif

#ifndef FALSE
# define FALSE                         (0U)
#endif

#ifndef __TMWTYPES__
#define __TMWTYPES__
#include <limits.h>

/*=======================================================================*
 * Target hardware information
 *   Device type: Intel->x86/Pentium
 *   Number of bits:     char:   8    short:   16    int:  32
 *                       long:  32      native word size:  32
 *   Byte ordering: LittleEndian
 *   Signed integer division rounds to: Zero
 *   Shift right on a signed integer as arithmetic shift: on
 *=======================================================================*/

/*=======================================================================*
 * Fixed width word size data types:                                     *
 *   int8_T, int16_T, int32_T     - signed 8, 16, or 32 bit integers     *
 *   uint8_T, uint16_T, uint32_T  - unsigned 8, 16, or 32 bit integers   *
 *   real32_T, real64_T           - 32 and 64 bit floating point numbers *
 *=======================================================================*/
typedef signed char int8_T;
typedef unsigned char uint8_T;
typedef short int16_T;
typedef unsigned short uint16_T;
typedef int int32_T;
typedef unsigned int uint32_T;
typedef float real32_T;
typedef double real64_T;

/*===========================================================================*
 * Generic type definitions: real_T, time_T, boolean_T, int_T, uint_T,       *
 *                           ulong_T, char_T and byte_T.                     *
 *===========================================================================*/
typedef double real_T;
typedef double time_T;
typedef unsigned char boolean_T;
typedef int int_T;
typedef unsigned int uint_T;
typedef unsigned long ulong_T;
typedef char char_T;
typedef unsigned char uchar_T;
typedef char_T byte_T;

/*=======================================================================*
 * Min and Max:                                                          *
 *   int8_T, int16_T, int32_T     - signed 8, 16, or 32 bit integers     *
 *   uint8_T, uint16_T, uint32_T  - unsigned 8, 16, or 32 bit integers   *
 *=======================================================================*/
#define MAX_int8_T                     ((int8_T)(127))
#define MIN_int8_T                     ((int8_T)(-128))
#define MAX_uint8_T                    ((uint8_T)(255U))
#define MIN_uint8_T                    ((uint8_T)(0U))
#define MAX_int16_T                    ((int16_T)(32767))
#define MIN_int16_T                    ((int16_T)(-32768))
#define MAX_uint16_T                   ((uint16_T)(65535U))
#define MIN_uint16_T                   ((uint16_T)(0U))
#define MAX_int32_T                    ((int32_T)(2147483647))
#define MIN_int32_T                    ((int32_T)(-2147483647-1))
#define MAX_uint32_T                   ((uint32_T)(0xFFFFFFFFU))
#define MIN_uint32_T                   ((uint32_T)(0U))

/* Logical type definitions */
#if (!defined(__cplusplus)) && (!defined(__true_false_are_keywords))
#  ifndef false
#   define false                       (0U)
#  endif

#  ifndef true
#   define true                        (1U)
#  endif
#endif

/*
 * Simulink Coder assumes the code is compiled on a target using a 2's complement representation
 * for signed integer values.
 */
#if ((SCHAR_MIN + 1) != -SCHAR_MAX)
#error "This code must be compiled using a 2's complement representation for signed integer values"
#endif

/* This ID is used to detect inclusion of an incompatible rtwtypes.h */
#define RTWTYPES_ID_C08S16I32L32N32F1
#else                                  /* __TMWTYPES__ */
#define TMWTYPES_PREVIOUSLY_INCLUDED
#endif                                 /* __TMWTYPES__ */

/* Block D-Work pointer type */
typedef void * pointer_T;

/* Simulink specific types */
#ifndef __SIMSTRUC_TYPES_H__
#define __SIMSTRUC_TYPES_H__

/* Trigger directions: falling, either, and rising */
typedef enum {
  FALLING_ZERO_CROSSING = -1,
  ANY_ZERO_CROSSING = 0,
  RISING_ZERO_CROSSING = 1
} ZCDirection;

/* Previous state of a trigger signal */
typedef uint8_T ZCSigState;

/* Initial value of a trigger zero crossing signal */
#define UNINITIALIZED_ZCSIG            0x03U
#define NEG_ZCSIG                      0x02U
#define POS_ZCSIG                      0x01U
#define ZERO_ZCSIG                     0x00U

/* Current state of a trigger signal */
typedef enum {
  FALLING_ZCEVENT = -1,
  NO_ZCEVENT = 0,
  RISING_ZCEVENT = 1
} ZCEventType;

#endif                                 /* __SIMSTRUC_TYPES_H__ */
#endif                                 /* __RTWTYPES_H__ */

#ifndef MIN
#define MIN(a,b)                       ((a) < (b) ? (a) : (b))
#endif

#ifndef MAX
#define MAX(a,b)                       ((a) > (b) ? (a) : (b))
#endif
#endif                                 /* RTW_HEADER_rtwtypes_h_ */
```

#### SimPID4.c
```c
/********************************************************************
 * COPYRIGHT -- Bernecker + Rainer Industrie-Elektronik Ges.m.b.H.
 ********************************************************************
 * Program: SimPID4
 * File: SimPID4.c
 * Author: 106001702
 * Created: Wed Nov 09 12:46:00 2011
 ********************************************************************
 * Implementation of program SimPID4
 ********************************************************************
 * Generated with B&R Automation Studio Target for Simulink V4.2
 * (ERT based)
 ********************************************************************/

#include "SimPID4.h"
#include "SimPID4_private.h"

/*  Defines */

/*  Data Types */

/**************************** GLOBAL DATA *************************************/
/*  Definitions */

/* Block signals (auto storage) */

/* Block states (auto storage) */

/*  Declarations  */

/***************************** FILE SCOPE DATA ********************************/

/*************************** FUNCTIONS ****************************************/

/* Model step function */
void SimPID4_step(struct SimPID4* inst)
{
  real_T rtb_Product;
  real_T rtb_Invertswitch;
  real32_T rtb_Product2;
  real32_T rtb_Gain2;
  real32_T rtb_SumI1;

  /* S-Function (bur_in): '<Root>/Input9' */
  inst->bur_SimPID4_B.Input9 = inst->mode;

  /* S-Function (bur_in): '<Root>/Input10' */
  inst->bur_SimPID4_B.Input10 = inst->u_man;

  /* S-Function (bur_in): '<Root>/Input6' */
  inst->bur_SimPID4_B.Input6 = inst->a;

  /* S-Function (bur_in): '<Root>/Input5' */
  inst->bur_SimPID4_B.Input5 = inst->invert;

  /* Switch: '<S2>/Invert switch' incorporates:
   *  Constant: '<S2>/Constant2'
   *  Constant: '<S2>/Constant3'
   */
  if (inst->bur_SimPID4_B.Input5) {
    rtb_Invertswitch = -1.0;
  } else {
    rtb_Invertswitch = 1.0;
  }

  /* End of Switch: '<S2>/Invert switch' */

  /* S-Function (bur_in): '<Root>/Input4' */
  inst->bur_SimPID4_B.Input4 = inst->w;

  /* Product: '<S2>/Product' incorporates:
   *  Constant: '<S2>/Scaling'
   */
  rtb_Product = 1.0 / (inst->wxmax - inst->wxmin) * (real_T)inst->bur_SimPID4_B.Input4;

  /* S-Function (bur_in): '<Root>/Input' */
  inst->bur_SimPID4_B.Input = inst->x;

  /* Sum: '<S2>/Sum' incorporates:
   *  Constant: '<S2>/Scaling'
   *  Product: '<S2>/Product1'
   */
  rtb_Product -= 1.0 / (inst->wxmax - inst->wxmin) * (real_T)inst->bur_SimPID4_B.Input;

  /* DeadZone: '<S2>/Deadband' */
  if (rtb_Product > inst->deadband) {
    rtb_Product -= inst->deadband;
  } else if (rtb_Product >= -inst->deadband) {
    rtb_Product = 0.0;
  } else {
    rtb_Product -= -inst->deadband;
  }

  /* End of DeadZone: '<S2>/Deadband' */

  /* Product: '<S2>/Product2' */
  rtb_Product2 = (real32_T)(rtb_Invertswitch * rtb_Product);

  /* Gain: '<S3>/Gain' */
  inst->bur_SimPID4_B.Gain = inst->P * rtb_Product2;

  /* S-Function (bur_in): '<Root>/Input1' */
  inst->bur_SimPID4_B.Input1 = inst->reset;

  /* S-Function (bur_in): '<Root>/Input2' */
  inst->bur_SimPID4_B.Input2 = inst->I0;

  /* DiscreteIntegrator: '<S3>/Integrator' */
  if (inst->bur_SimPID4_DWork.Integrator_IC_LOADING != 0) {
    inst->bur_SimPID4_DWork.Integrator_DSTATE = inst->bur_SimPID4_B.Input2;
  }

  if (inst->bur_SimPID4_B.Input1) {
    inst->bur_SimPID4_DWork.Integrator_DSTATE = inst->bur_SimPID4_B.Input2;
  }

  inst->bur_SimPID4_B.Integrator = inst->bur_SimPID4_DWork.Integrator_DSTATE;

  /* End of DiscreteIntegrator: '<S3>/Integrator' */

  /* Gain: '<S3>/Gain2' */
  rtb_Gain2 = inst->D * rtb_Product2;

  /* S-Function (bur_in): '<Root>/Input3' */
  inst->bur_SimPID4_B.Input3 = inst->D0;

  /* DiscreteIntegrator: '<S3>/Filter' */
  if (inst->bur_SimPID4_DWork.Filter_IC_LOADING != 0) {
    inst->bur_SimPID4_DWork.Filter_DSTATE = inst->bur_SimPID4_B.Input3;
  }

  if (inst->bur_SimPID4_B.Input1) {
    inst->bur_SimPID4_DWork.Filter_DSTATE = inst->bur_SimPID4_B.Input3;
  }

  /* End of DiscreteIntegrator: '<S3>/Filter' */

  /* Gain: '<S3>/Filter Coefficient' incorporates:
   *  DiscreteIntegrator: '<S3>/Filter'
   *  Sum: '<S3>/SumD'
   */
  inst->bur_SimPID4_B.FilterCoefficient = (rtb_Gain2 - inst->bur_SimPID4_DWork.Filter_DSTATE) * inst->N;

  /* Sum: '<S3>/Sum2' incorporates:
   *  Sum: '<S3>/Sum1'
   */
  rtb_Gain2 = ((inst->bur_SimPID4_B.Gain + inst->bur_SimPID4_B.Integrator) +
               inst->bur_SimPID4_B.FilterCoefficient) + inst->bur_SimPID4_B.Input6;

  /* Saturate: '<S3>/Saturation' */
  inst->bur_SimPID4_B.Saturation = rtb_Gain2 >= inst->umax ? inst->umax : rtb_Gain2 <= inst->umin ? inst->umin :
    rtb_Gain2;

  /* MultiPortSwitch: '<S2>/Mode switch' */
  switch (inst->bur_SimPID4_B.Input9) {
   case 1:
    inst->bur_SimPID4_B.Modeswitch = inst->bur_SimPID4_B.Input10;
    break;

   case 2:
    inst->bur_SimPID4_B.Modeswitch = inst->bur_SimPID4_B.Input10;
    break;

   default:
    inst->bur_SimPID4_B.Modeswitch = inst->bur_SimPID4_B.Saturation;
    break;
  }

  /* End of MultiPortSwitch: '<S2>/Mode switch' */

  /* S-Function (bur_out): '<Root>/Output' */
  inst->u = inst->bur_SimPID4_B.Modeswitch;

  /* S-Function (bur_out): '<Root>/Output1' */
  inst->up = inst->bur_SimPID4_B.Gain;

  /* S-Function (bur_out): '<Root>/Output2' */
  inst->ui = inst->bur_SimPID4_B.Integrator;

  /* S-Function (bur_out): '<Root>/Output3' */
  inst->ud = inst->bur_SimPID4_B.FilterCoefficient;

  /* S-Function (bur_out): '<Root>/Output4' */
  inst->u_tr = inst->bur_SimPID4_B.Saturation;

  /* S-Function (bur_in): '<Root>/Input7' */
  inst->bur_SimPID4_B.Input7 = inst->fbk_mode;

  /* S-Function (bur_in): '<Root>/Input8' */
  inst->bur_SimPID4_B.Input8 = inst->u_fbk;

  /* MultiPortSwitch: '<S3>/Multiport Switch' */
  if (inst->bur_SimPID4_B.Input7 == 1) {
    rtb_SumI1 = inst->bur_SimPID4_B.Input8;
  } else {
    rtb_SumI1 = inst->bur_SimPID4_B.Saturation;
  }

  /* End of MultiPortSwitch: '<S3>/Multiport Switch' */

  /* Sum: '<S4>/Sum' */
  rtb_Gain2 = rtb_SumI1 - rtb_Gain2;

  /* MultiPortSwitch: '<S2>/Tracking switch' incorporates:
   *  Constant: '<S2>/Constant'
   *  Constant: '<S2>/Constant1'
   */
  switch (inst->bur_SimPID4_B.Input9) {
   case 1:
    rtb_Invertswitch = 0.0;
    break;

   case 2:
    rtb_Invertswitch = inst->Kt;
    break;

   default:
    rtb_Invertswitch = 0.0;
    break;
  }

  /* End of MultiPortSwitch: '<S2>/Tracking switch' */

  /* Sum: '<S3>/SumI1' incorporates:
   *  Gain: '<S3>/Gain1'
   *  Product: '<S3>/Product'
   *  Sum: '<S3>/SumI3'
   */
  rtb_SumI1 = (real32_T)((real_T)(inst->bur_SimPID4_B.Input10 - inst->bur_SimPID4_B.Saturation) *
    rtb_Invertswitch) + inst->I * rtb_Product2;

  /* Switch: '<S3>/Switch' incorporates:
   *  Abs: '<S4>/Abs'
   *  Constant: '<S3>/Constant4'
   *  Constant: '<S5>/Constant'
   *  Logic: '<S4>/AND'
   *  RelationalOperator: '<S4>/Equal'
   *  RelationalOperator: '<S5>/Compare'
   *  Signum: '<S4>/SignPreIntegrator'
   *  Signum: '<S4>/SignPreSat'
   */
  if (((real32_T)fabs(rtb_Gain2) > 0.005F) && ((rtb_Gain2 < 0.0F ? -1.0F :
        rtb_Gain2 > 0.0F ? 1.0F : rtb_Gain2) != (rtb_SumI1 < 0.0F ? -1.0F :
        rtb_SumI1 > 0.0F ? 1.0F : rtb_SumI1))) {
    rtb_SumI1 = 0.0F;
  }

  /* End of Switch: '<S3>/Switch' */

  /* Update for DiscreteIntegrator: '<S3>/Integrator' */
  inst->bur_SimPID4_DWork.Integrator_IC_LOADING = 0U;
  inst->bur_SimPID4_DWork.Integrator_DSTATE = 0.01F * rtb_SumI1 +
    inst->bur_SimPID4_DWork.Integrator_DSTATE;

  /* Update for DiscreteIntegrator: '<S3>/Filter' */
  inst->bur_SimPID4_DWork.Filter_IC_LOADING = 0U;
  inst->bur_SimPID4_DWork.Filter_DSTATE = 0.01F * inst->bur_SimPID4_B.FilterCoefficient +
    inst->bur_SimPID4_DWork.Filter_DSTATE;
}

/* Model initialize function */
void SimPID4_initialize(struct SimPID4* inst)
{
  /* InitializeConditions for DiscreteIntegrator: '<S3>/Integrator' */
  inst->bur_SimPID4_DWork.Integrator_IC_LOADING = 1U;

  /* InitializeConditions for DiscreteIntegrator: '<S3>/Filter' */
  inst->bur_SimPID4_DWork.Filter_IC_LOADING = 1U;
}

/* Model terminate function */
void SimPID4_terminate(struct SimPID4* inst)
{
  /* (no terminate code required) */
}

/*======================== TOOL VERSION INFORMATION ==========================*
 * MATLAB 7.12 (R2011a)09-Mar-2011                                            *
 * Simulink 7.7 (R2011a)09-Mar-2011                                           *
 * Simulink Coder 8.0 (R2011a)09-Mar-2011                                     *
 * Embedded Coder 6.0 (R2011a)09-Mar-2011                                     *
 * Stateflow 7.7 (R2011a)09-Mar-2011                                          *
 * Simulink Fixed Point 6.5 (R2011a)09-Mar-2011                               *
 *============================================================================*/

/*======================= LICENSE IN USE INFORMATION =========================*
 * matlab                                                                     *
 * matlab_coder                                                               *
 * real-time_workshop                                                         *
 * rtw_embedded_coder                                                         *
 * simulink                                                                   *
 *============================================================================*/
```

#### main.c
```c
/********************************************************************
 * COPYRIGHT -- Bernecker + Rainer Industrie-Elektronik Ges.m.b.H.
 ********************************************************************
 * Program: SimPID4
 * File: main.c
 * Author: 106001702
 * Created: Wed Nov 09 12:46:00 2011
 ********************************************************************
 * Implementation of program SimPID4
 ********************************************************************
 * Generated with B&R Automation Studio Target for Simulink V4.2
 * (ERT based)
 ********************************************************************/

#include <bur/plctypes.h>
#include "SimPID4.h"
#include "rtwtypes.h"

BOOL bur_firsttime = TRUE;

/*  Defines */
#define SS_TERMINATE 4
#define SS_OUTPUT 3
#define SS_INITIALIZE 2

/*  Data Types */

/**************************** GLOBAL DATA *************************************/
/*  Definitions */

/*  Declarations  */

/***************************** FILE SCOPE DATA ********************************/

/*************************** FUNCTIONS ****************************************/
#ifdef __cplusplus

unsigned long bur_heap_size = 6553500;

#endif

void SimPID4(struct SimPID4* inst)
{
  switch (inst->ssMethodType)
  {
   case SS_INITIALIZE:
    /* call model initialize function */
    SimPID4_initialize(inst);
    break;

   case SS_OUTPUT:
    /* call model step function */
    SimPID4_step(inst);

    break;

   case SS_TERMINATE:
    /* call model terminate function */
    SimPID4_terminate(inst);
    break;
  }
}

/*****************************************************************************
   Function block sample time: 0.01s
 *****************************************************************************/

/*****************************************************************************
   B&R Automation Studio Target for Simulink Version: A4.2.11 (15-Jan-2014)
 *****************************************************************************/

/*======================== TOOL VERSION INFORMATION ==========================*
 * MATLAB 7.12 (R2011a)09-Mar-2011                                            *
 * Simulink 7.7 (R2011a)09-Mar-2011                                           *
 * Simulink Coder 8.0 (R2011a)09-Mar-2011                                     *
 * Embedded Coder 6.0 (R2011a)09-Mar-2011                                     *
 * Stateflow 7.7 (R2011a)09-Mar-2011                                          *
 * Simulink Fixed Point 6.5 (R2011a)09-Mar-2011                               *
 *============================================================================*/

/*======================= LICENSE IN USE INFORMATION =========================*
 * matlab                                                                     *
 * matlab_coder                                                               *
 * real-time_workshop                                                         *
 * rtw_embedded_coder                                                         *
 * simulink                                                                   *
 *============================================================================*/
```

#### lib_properties.txt
```
For manual assignment to hardware configuration please
add the following additional include directories:

\Logical\MATLAB_includes\R2011a\

And the following additional build options:

-lm -D MODEL=SimPID4 -D NUMST=1 -D NCSTATES=0 -D HAVESTDIO -D ONESTEPFCN=1 -D TERMFCN=1 -D MAT_FILE=0 -D MULTI_INSTANCE_CODE=0 -D INTEGER_CODE=0 -D MT=0 -D TID01EQ=0
```

### Library Logical/Libraries/lSim3pCTR (ANSIC)

#### lSim3pCTR.fun
```iecst
FUNCTION_BLOCK Sim3pCTR
  VAR_INPUT
    ssMethodType: SINT;
  END_VAR  VAR_INPUT
        Enable : BOOL := FALSE; (**)
  END_VAR
  VAR_INPUT
        SetValue : REAL; (*Set Value*)
  END_VAR
  VAR_INPUT
        HysPos : REAL; (*positive hysteresis for trigger value*)
  END_VAR
  VAR_INPUT
        HysNeg : REAL; (*negative hysteresis for trigger value*)
  END_VAR
  VAR_INPUT
        ActValue : REAL; (*actual value*)
  END_VAR
  VAR_INPUT
        dY_up : REAL; (*positive gradient*)
  END_VAR
  VAR_INPUT
        dY_down : REAL; (*negative gradient*)
  END_VAR
  VAR_INPUT
        CycleTime : REAL; (*cycle time in which FUB is used*)
  END_VAR
  VAR_INPUT
        Reset : BOOL := FALSE; (*reset bit*)
  END_VAR
  VAR_INPUT
        InitValue : REAL; (*initial value when reset bit is set*)
  END_VAR
  VAR_INPUT
        bInverse : BOOL := FALSE; (*Invert actuating direction of controller*)
  END_VAR
  VAR_INPUT
        bRamp_Y_min : BOOL := FALSE; (*ramp output y to minimum*)
  END_VAR
  VAR_INPUT
        bRamp_Y_max : BOOL := FALSE; (*ramp output y to maximum*)
  END_VAR
  VAR_INPUT
        Y_min : REAL; (*minimal Limit for Output Y*)
  END_VAR
  VAR_INPUT
        Y_max : REAL; (*maximal Limit for Output Y*)
  END_VAR
  VAR_OUTPUT
        Y : REAL; (*Controller Output*)
  END_VAR
  VAR_OUTPUT
        bY_min_limit : BOOL := FALSE; (*Y is in minimum limitation*)
  END_VAR
  VAR_OUTPUT
        bY_max_limit : BOOL := FALSE; (*Y is in maximum limitation*)
  END_VAR
  VAR_OUTPUT
        State : INT; (*state::
0: steady
1: decrease
2: increase*)
  END_VAR
	VAR
		bur_Sim3pCTR_DWork : D_Work_Sim3pCTR;
	END_VAR
	VAR
		bur_Sim3pCTR_B : BlockIO_Sim3pCTR;
	END_VAR
END_FUNCTION_BLOCK
```

#### lSim3pCTR.typ
```iecst
TYPE
	D_Work_Sim3pCTR : STRUCT

		UnitDelay_DSTATE : REAL;
		is_active_c1_Sim3pCTR : USINT;
		is_c1_Sim3pCTR : USINT;
		is_enabled : USINT;
		is_manual_ramp : USINT;
		is_normal : USINT;
		is_inverse : USINT;
	END_STRUCT;

	 BlockIO_Sim3pCTR : STRUCT

		Input9 : REAL;
		Input1 : REAL;
		Input2 : REAL;
		Input3 : REAL;
		Input4 : REAL;
		Input5 : REAL;
		Input6 : REAL;
		Input8 : REAL;
		Input10 : REAL;
		Input11 : REAL;
		Switch2 : REAL;
		state : INT;
		Input : BOOL;
		Input7 : BOOL;
		Input14 : BOOL;
		Input12 : BOOL;
		Input13 : BOOL;
		RelationalOperator : BOOL;
		RelationalOperator1 : BOOL;
	END_STRUCT;

END_TYPE
```

#### lSim3pCTR.var
```iecst
VAR CONSTANT
    SS_INITIALIZE: SINT := 2; (* initialize function block *)
    SS_OUTPUT: SINT := 3; (* run function block cyclically *)
    SS_TERMINATE: SINT := 4; (* terminate function block *)
END_VAR
```

#### Sim3pCTR.h
```c
/********************************************************************
 * COPYRIGHT -- Bernecker + Rainer Industrie-Elektronik Ges.m.b.H.
 ********************************************************************
 * Program: Sim3pCTR
 * File: Sim3pCTR.h
 * Author: 105051472
 * Created: Thu Jan 10 08:03:20 2013
 ********************************************************************
 * Header for program Sim3pCTR
 ********************************************************************
 * Generated with B&R Automation Studio Target for Simulink V3.3
 * (ERT based)
 ********************************************************************/

#ifndef RTW_HEADER_Sim3pCTR_h_
#define RTW_HEADER_Sim3pCTR_h_
#ifndef Sim3pCTR_COMMON_INCLUDES_
# define Sim3pCTR_COMMON_INCLUDES_
#include "rtwtypes.h"
#endif                                 /* Sim3pCTR_COMMON_INCLUDES_ */

#include "Sim3pCTR_types.h"
#include "lSim3pCTR.h"

/* Macros for accessing real-time model data structure */
#ifndef rtmGetErrorStatus
# define rtmGetErrorStatus(rtm)        ((void*) 0)
#endif

#ifndef rtmSetErrorStatus
# define rtmSetErrorStatus(rtm, val)   ((void) 0)
#endif

#ifndef rtmGetStopRequested
# define rtmGetStopRequested(rtm)      ((void*) 0)
#endif

#ifndef MIN
#define MIN(a,b)                       ((a) < (b) ? (a) : (b))
#endif

#ifndef MAX
#define MAX(a,b)                       ((a) > (b) ? (a) : (b))
#endif

/* Block signals (auto storage) */

/* Block states (auto storage) for system '<Root>' */

/* Block signals (auto storage) */
extern BlockIO_Sim3pCTR Sim3pCTR_B;

/* Block states (auto storage) */
extern D_Work_Sim3pCTR Sim3pCTR_DWork;

/* Model entry point functions */
extern void Sim3pCTR_initialize(struct Sim3pCTR* inst);
extern void Sim3pCTR_step(struct Sim3pCTR* inst);
extern void Sim3pCTR_terminate(struct Sim3pCTR* inst);

/*-
 * The generated code includes comments that allow you to trace directly
 * back to the appropriate location in the model.  The basic format
 * is <system>/block_name, where system is the system number (uniquely
 * assigned by Simulink) and block_name is the name of the block.
 *
 * Use the MATLAB hilite_system command to trace the generated code back
 * to the model.  For example,
 *
 * hilite_system('<S3>')    - opens system 3
 * hilite_system('<S3>/Kp') - opens and selects block Kp which resides in S3
 *
 * Here is the system hierarchy for this model
 *
 * '<Root>' : Sim3pCTR
 * '<S1>'   : Sim3pCTR/Model Info
 * '<S2>'   : Sim3pCTR/Sim3pCTR
 * '<S3>'   : Sim3pCTR/Sim3pCTR/Integrator
 * '<S4>'   : Sim3pCTR/Sim3pCTR/StateMachine
 * '<S5>'   : Sim3pCTR/Sim3pCTR/Integrator/Saturation Dynamic
 */
#endif                                 /* RTW_HEADER_Sim3pCTR_h_ */
```

#### Sim3pCTR_private.h
```c
/********************************************************************
 * COPYRIGHT -- Bernecker + Rainer Industrie-Elektronik Ges.m.b.H.
 ********************************************************************
 * Program: Sim3pCTR
 * File: Sim3pCTR_private.h
 * Author: 105051472
 * Created: Thu Jan 10 08:03:20 2013
 ********************************************************************
 * Header for program Sim3pCTR
 ********************************************************************
 * Generated with B&R Automation Studio Target for Simulink V3.3
 * (ERT based)
 ********************************************************************/

#ifndef RTW_HEADER_Sim3pCTR_private_h_
#define RTW_HEADER_Sim3pCTR_private_h_
#include "rtwtypes.h"
#include <bur/plctypes.h>
#define CALL_EVENT                     (-1)
#ifndef __RTWTYPES_H__
#error This file requires rtwtypes.h to be included
#else
#ifdef TMWTYPES_PREVIOUSLY_INCLUDED
#error This file requires rtwtypes.h to be included before tmwtypes.h
#else

/* Check for inclusion of an incorrect version of rtwtypes.h */
#ifndef RTWTYPES_ID_C08S16I32L32N32F1
#error This code was generated with a different "rtwtypes.h" than the file included
#endif                                 /* RTWTYPES_ID_C08S16I32L32N32F1 */
#endif                                 /* TMWTYPES_PREVIOUSLY_INCLUDED */
#endif                                 /* __RTWTYPES_H__ */

#ifndef MIN
#define MIN(a,b)                       ((a) < (b) ? (a) : (b))
#endif

#ifndef MAX
#define MAX(a,b)                       ((a) > (b) ? (a) : (b))
#endif
#endif                                 /* RTW_HEADER_Sim3pCTR_private_h_ */
```

#### Sim3pCTR_types.h
```c
/********************************************************************
 * COPYRIGHT -- Bernecker + Rainer Industrie-Elektronik Ges.m.b.H.
 ********************************************************************
 * Program: Sim3pCTR
 * File: Sim3pCTR_types.h
 * Author: 105051472
 * Created: Thu Jan 10 08:03:20 2013
 ********************************************************************
 * Header for program Sim3pCTR
 ********************************************************************
 * Generated with B&R Automation Studio Target for Simulink V3.3
 * (ERT based)
 ********************************************************************/

#ifndef RTW_HEADER_Sim3pCTR_types_h_
#define RTW_HEADER_Sim3pCTR_types_h_
#ifndef MIN
#define MIN(a,b)                       ((a) < (b) ? (a) : (b))
#endif

#ifndef MAX
#define MAX(a,b)                       ((a) > (b) ? (a) : (b))
#endif
#endif                                 /* RTW_HEADER_Sim3pCTR_types_h_ */
```

#### rtwtypes.h
```c
/********************************************************************
 * COPYRIGHT -- Bernecker + Rainer Industrie-Elektronik Ges.m.b.H.
 ********************************************************************
 * Program: Sim3pCTR
 * File: rtwtypes.h
 * Author: 105051472
 * Created: Thu Jan 10 08:03:20 2013
 ********************************************************************
 * Header for program Sim3pCTR
 ********************************************************************
 * Generated with B&R Automation Studio Target for Simulink V3.3
 * (ERT based)
 ********************************************************************/

#ifndef RTW_HEADER_rtwtypes_h_
#define RTW_HEADER_rtwtypes_h_
#ifndef __RTWTYPES_H__
#define __RTWTYPES_H__
#ifndef TRUE
# define TRUE                          (1U)
#endif

#ifndef FALSE
# define FALSE                         (0U)
#endif

#ifndef __TMWTYPES__
#define __TMWTYPES__
#include <limits.h>

/*=======================================================================*
 * Target hardware information
 *   Device type: Intel->x86/Pentium
 *   Number of bits:     char:   8    short:   16    int:  32
 *                       long:  32      native word size:  32
 *   Byte ordering: LittleEndian
 *   Signed integer division rounds to: Zero
 *   Shift right on a signed integer as arithmetic shift: on
 *=======================================================================*/

/*=======================================================================*
 * Fixed width word size data types:                                     *
 *   int8_T, int16_T, int32_T     - signed 8, 16, or 32 bit integers     *
 *   uint8_T, uint16_T, uint32_T  - unsigned 8, 16, or 32 bit integers   *
 *   real32_T, real64_T           - 32 and 64 bit floating point numbers *
 *=======================================================================*/
typedef signed char int8_T;
typedef unsigned char uint8_T;
typedef short int16_T;
typedef unsigned short uint16_T;
typedef int int32_T;
typedef unsigned int uint32_T;
typedef float real32_T;
typedef double real64_T;

/*===========================================================================*
 * Generic type definitions: real_T, time_T, boolean_T, int_T, uint_T,       *
 *                           ulong_T, char_T and byte_T.                     *
 *===========================================================================*/
typedef double real_T;
typedef double time_T;
typedef unsigned char boolean_T;
typedef int int_T;
typedef unsigned int uint_T;
typedef unsigned long ulong_T;
typedef char char_T;
typedef unsigned char uchar_T;
typedef char_T byte_T;

/*=======================================================================*
 * Min and Max:                                                          *
 *   int8_T, int16_T, int32_T     - signed 8, 16, or 32 bit integers     *
 *   uint8_T, uint16_T, uint32_T  - unsigned 8, 16, or 32 bit integers   *
 *=======================================================================*/
#define MAX_int8_T                     ((int8_T)(127))
#define MIN_int8_T                     ((int8_T)(-128))
#define MAX_uint8_T                    ((uint8_T)(255U))
#define MIN_uint8_T                    ((uint8_T)(0U))
#define MAX_int16_T                    ((int16_T)(32767))
#define MIN_int16_T                    ((int16_T)(-32768))
#define MAX_uint16_T                   ((uint16_T)(65535U))
#define MIN_uint16_T                   ((uint16_T)(0U))
#define MAX_int32_T                    ((int32_T)(2147483647))
#define MIN_int32_T                    ((int32_T)(-2147483647-1))
#define MAX_uint32_T                   ((uint32_T)(0xFFFFFFFFU))
#define MIN_uint32_T                   ((uint32_T)(0U))

/* Logical type definitions */
#if (!defined(__cplusplus)) && (!defined(__true_false_are_keywords))
#  ifndef false
#   define false                       (0U)
#  endif

#  ifndef true
#   define true                        (1U)
#  endif
#endif

/*
 * Simulink Coder assumes the code is compiled on a target using a 2's complement representation
 * for signed integer values.
 */
#if ((SCHAR_MIN + 1) != -SCHAR_MAX)
#error "This code must be compiled using a 2's complement representation for signed integer values"
#endif

/* This ID is used to detect inclusion of an incompatible rtwtypes.h */
#define RTWTYPES_ID_C08S16I32L32N32F1
#else                                  /* __TMWTYPES__ */
#define TMWTYPES_PREVIOUSLY_INCLUDED
#endif                                 /* __TMWTYPES__ */

/* Block D-Work pointer type */
typedef void * pointer_T;

/* Simulink specific types */
#ifndef __SIMSTRUC_TYPES_H__
#define __SIMSTRUC_TYPES_H__

/* Trigger directions: falling, either, and rising */
typedef enum {
  FALLING_ZERO_CROSSING = -1,
  ANY_ZERO_CROSSING = 0,
  RISING_ZERO_CROSSING = 1
} ZCDirection;

/* Previous state of a trigger signal */
typedef uint8_T ZCSigState;

/* Initial value of a trigger zero crossing signal */
#define UNINITIALIZED_ZCSIG            0x03U
#define NEG_ZCSIG                      0x02U
#define POS_ZCSIG                      0x01U
#define ZERO_ZCSIG                     0x00U

/* Current state of a trigger signal */
typedef enum {
  FALLING_ZCEVENT = -1,
  NO_ZCEVENT = 0,
  RISING_ZCEVENT = 1
} ZCEventType;

#endif                                 /* __SIMSTRUC_TYPES_H__ */
#endif                                 /* __RTWTYPES_H__ */

#ifndef MIN
#define MIN(a,b)                       ((a) < (b) ? (a) : (b))
#endif

#ifndef MAX
#define MAX(a,b)                       ((a) > (b) ? (a) : (b))
#endif
#endif                                 /* RTW_HEADER_rtwtypes_h_ */
```

#### Sim3pCTR.c
```c
/********************************************************************
 * COPYRIGHT -- Bernecker + Rainer Industrie-Elektronik Ges.m.b.H.
 ********************************************************************
 * Program: Sim3pCTR
 * File: Sim3pCTR.c
 * Author: 105051472
 * Created: Thu Jan 10 08:03:20 2013
 ********************************************************************
 * Implementation of program Sim3pCTR
 ********************************************************************
 * Generated with B&R Automation Studio Target for Simulink V3.3
 * (ERT based)
 ********************************************************************/

#include "Sim3pCTR.h"
#include "Sim3pCTR_private.h"

/*  Defines */

/* Named constants for Stateflow: '<S2>/StateMachine' */
#define Sim3pCTR_IN_NO_ACTIVE_CHILD    (0U)
#define Sim3pCTR_IN_decrease           (1U)
#define Sim3pCTR_IN_decrease_inv       (1U)
#define Sim3pCTR_IN_disabled           (1U)
#define Sim3pCTR_IN_enabled            (2U)
#define Sim3pCTR_IN_increase           (2U)
#define Sim3pCTR_IN_increase_inv       (2U)
#define Sim3pCTR_IN_inverse            (1U)
#define Sim3pCTR_IN_man_decrease       (1U)
#define Sim3pCTR_IN_man_increase       (2U)
#define Sim3pCTR_IN_man_steady         (3U)
#define Sim3pCTR_IN_manual_ramp        (3U)
#define Sim3pCTR_IN_normal             (2U)
#define Sim3pCTR_IN_steady             (3U)
#define Sim3pCTR_IN_steady_inv         (3U)

/*  Data Types */

/**************************** GLOBAL DATA *************************************/
/*  Definitions */

/* Block signals (auto storage) */

/* Block states (auto storage) */

/*  Declarations  */

/***************************** FILE SCOPE DATA ********************************/

/*************************** FUNCTIONS ****************************************/

/* Model step function */
void Sim3pCTR_step(struct Sim3pCTR* inst)
{
  real32_T rtb_Switch;
  real32_T rtb_Add;
  real32_T rtb_Add1;

  /* S-Function (bur_in): '<Root>/Input' */
  inst->bur_Sim3pCTR_B.Input = inst->Enable;

  /* S-Function (bur_in): '<Root>/Input9' */
  inst->bur_Sim3pCTR_B.Input9 = inst->SetValue;

  /* S-Function (bur_in): '<Root>/Input1' */
  inst->bur_Sim3pCTR_B.Input1 = inst->HysPos;

  /* S-Function (bur_in): '<Root>/Input2' */
  inst->bur_Sim3pCTR_B.Input2 = inst->HysNeg;

  /* S-Function (bur_in): '<Root>/Input3' */
  inst->bur_Sim3pCTR_B.Input3 = inst->ActValue;

  /* S-Function (bur_in): '<Root>/Input4' */
  inst->bur_Sim3pCTR_B.Input4 = inst->dY_up;

  /* S-Function (bur_in): '<Root>/Input5' */
  inst->bur_Sim3pCTR_B.Input5 = inst->dY_down;

  /* S-Function (bur_in): '<Root>/Input6' */
  inst->bur_Sim3pCTR_B.Input6 = inst->CycleTime;

  /* S-Function (bur_in): '<Root>/Input7' */
  inst->bur_Sim3pCTR_B.Input7 = inst->Reset;

  /* S-Function (bur_in): '<Root>/Input8' */
  inst->bur_Sim3pCTR_B.Input8 = inst->InitValue;

  /* S-Function (bur_in): '<Root>/Input14' */
  inst->bur_Sim3pCTR_B.Input14 = inst->bInverse;

  /* S-Function (bur_in): '<Root>/Input12' */
  inst->bur_Sim3pCTR_B.Input12 = inst->bRamp_Y_min;

  /* S-Function (bur_in): '<Root>/Input13' */
  inst->bur_Sim3pCTR_B.Input13 = inst->bRamp_Y_max;

  /* S-Function (bur_in): '<Root>/Input10' */
  inst->bur_Sim3pCTR_B.Input10 = inst->Y_min;

  /* S-Function (bur_in): '<Root>/Input11' */
  inst->bur_Sim3pCTR_B.Input11 = inst->Y_max;

  /* Outputs for Atomic SubSystem: '<Root>/Sim3pCTR' */
  /* Sum: '<S2>/Add' */
  rtb_Add = inst->bur_Sim3pCTR_B.Input9 + inst->bur_Sim3pCTR_B.Input1;

  /* Sum: '<S2>/Add1' */
  rtb_Add1 = inst->bur_Sim3pCTR_B.Input9 - inst->bur_Sim3pCTR_B.Input2;

  /* Switch: '<S3>/Switch' incorporates:
   *  UnitDelay: '<S3>/Unit Delay'
   */
  if (inst->bur_Sim3pCTR_B.Input7) {
    rtb_Switch = inst->bur_Sim3pCTR_B.Input8;
  } else {
    rtb_Switch = inst->bur_Sim3pCTR_DWork.UnitDelay_DSTATE;
  }

  /* End of Switch: '<S3>/Switch' */

  /* Switch: '<S5>/Switch2' incorporates:
   *  RelationalOperator: '<S5>/LowerRelop1'
   */
  if (rtb_Switch > inst->bur_Sim3pCTR_B.Input11) {
    inst->bur_Sim3pCTR_B.Switch2 = inst->bur_Sim3pCTR_B.Input11;
  } else {
    /* Switch: '<S5>/Switch' incorporates:
     *  RelationalOperator: '<S5>/UpperRelop'
     */
    if (rtb_Switch < inst->bur_Sim3pCTR_B.Input10) {
      inst->bur_Sim3pCTR_B.Switch2 = inst->bur_Sim3pCTR_B.Input10;
    } else {
      inst->bur_Sim3pCTR_B.Switch2 = rtb_Switch;
    }

    /* End of Switch: '<S5>/Switch' */
  }

  /* End of Switch: '<S5>/Switch2' */

  /* RelationalOperator: '<S2>/Relational Operator' */
  inst->bur_Sim3pCTR_B.RelationalOperator = ((inst->bur_Sim3pCTR_B.Switch2 <= inst->bur_Sim3pCTR_B.Input10));

  /* RelationalOperator: '<S2>/Relational Operator1' */
  inst->bur_Sim3pCTR_B.RelationalOperator1 = ((inst->bur_Sim3pCTR_B.Switch2 >= inst->bur_Sim3pCTR_B.Input11));

  /* Stateflow: '<S2>/StateMachine' */

  /* Gateway: Sim3pCTR/StateMachine */
  /* During: Sim3pCTR/StateMachine */
  if (inst->bur_Sim3pCTR_DWork.is_active_c1_Sim3pCTR == 0) {
    /* Entry: Sim3pCTR/StateMachine */
    inst->bur_Sim3pCTR_DWork.is_active_c1_Sim3pCTR = 1U;

    /* Transition: '<S4>:79' */
    inst->bur_Sim3pCTR_DWork.is_c1_Sim3pCTR = Sim3pCTR_IN_disabled;

    /* Entry 'disabled': '<S4>:69' */
    inst->bur_Sim3pCTR_B.state = 0;
  } else {
    switch (inst->bur_Sim3pCTR_DWork.is_c1_Sim3pCTR) {
     case Sim3pCTR_IN_disabled:
      /* During 'disabled': '<S4>:69' */
      if (inst->bur_Sim3pCTR_B.Input == TRUE) {
        /* Transition: '<S4>:70' */
        inst->bur_Sim3pCTR_DWork.is_c1_Sim3pCTR = Sim3pCTR_IN_enabled;

        /* Transition: '<S4>:123' */
        inst->bur_Sim3pCTR_DWork.is_enabled = Sim3pCTR_IN_normal;

        /* Transition: '<S4>:78' */
        inst->bur_Sim3pCTR_DWork.is_normal = Sim3pCTR_IN_steady;

        /* Entry 'steady': '<S4>:11' */
        inst->bur_Sim3pCTR_B.state = 0;
      }
      break;

     case Sim3pCTR_IN_enabled:
      /* During 'enabled': '<S4>:62' */
      if (inst->bur_Sim3pCTR_B.Input == FALSE) {
        /* Transition: '<S4>:71' */
        inst->bur_Sim3pCTR_DWork.is_inverse = (uint8_T)Sim3pCTR_IN_NO_ACTIVE_CHILD;
        inst->bur_Sim3pCTR_DWork.is_enabled = (uint8_T)Sim3pCTR_IN_NO_ACTIVE_CHILD;
        inst->bur_Sim3pCTR_DWork.is_normal = (uint8_T)Sim3pCTR_IN_NO_ACTIVE_CHILD;
        inst->bur_Sim3pCTR_DWork.is_c1_Sim3pCTR = Sim3pCTR_IN_disabled;

        /* Entry 'disabled': '<S4>:69' */
        inst->bur_Sim3pCTR_B.state = 0;
      } else if (inst->bur_Sim3pCTR_B.Input13 || inst->bur_Sim3pCTR_B.Input12) {
        /* Transition: '<S4>:99' */
        inst->bur_Sim3pCTR_DWork.is_inverse = (uint8_T)Sim3pCTR_IN_NO_ACTIVE_CHILD;
        inst->bur_Sim3pCTR_DWork.is_enabled = (uint8_T)Sim3pCTR_IN_NO_ACTIVE_CHILD;
        inst->bur_Sim3pCTR_DWork.is_normal = (uint8_T)Sim3pCTR_IN_NO_ACTIVE_CHILD;
        inst->bur_Sim3pCTR_DWork.is_c1_Sim3pCTR = Sim3pCTR_IN_manual_ramp;

        /* Transition: '<S4>:87' */
        inst->bur_Sim3pCTR_DWork.is_manual_ramp = Sim3pCTR_IN_man_steady;

        /* Entry 'man_steady': '<S4>:88' */
        inst->bur_Sim3pCTR_B.state = 0;
      } else {
        switch (inst->bur_Sim3pCTR_DWork.is_enabled) {
         case Sim3pCTR_IN_inverse:
          /* During 'inverse': '<S4>:109' */
          if (inst->bur_Sim3pCTR_B.Input14 == FALSE) {
            /* Transition: '<S4>:121' */
            inst->bur_Sim3pCTR_DWork.is_inverse = (uint8_T)Sim3pCTR_IN_NO_ACTIVE_CHILD;
            inst->bur_Sim3pCTR_DWork.is_enabled = Sim3pCTR_IN_normal;

            /* Transition: '<S4>:78' */
            inst->bur_Sim3pCTR_DWork.is_normal = Sim3pCTR_IN_steady;

            /* Entry 'steady': '<S4>:11' */
            inst->bur_Sim3pCTR_B.state = 0;
          } else {
            switch (inst->bur_Sim3pCTR_DWork.is_inverse) {
             case Sim3pCTR_IN_decrease_inv:
              /* During 'decrease_inv': '<S4>:117' */
              if ((inst->bur_Sim3pCTR_B.Input3 <= inst->bur_Sim3pCTR_B.Input9) ||
                  inst->bur_Sim3pCTR_B.RelationalOperator1) {
                /* Transition: '<S4>:112' */
                inst->bur_Sim3pCTR_DWork.is_inverse = Sim3pCTR_IN_steady_inv;

                /* Entry 'steady_inv': '<S4>:115' */
                inst->bur_Sim3pCTR_B.state = 0;
              }
              break;

             case Sim3pCTR_IN_increase_inv:
              /* During 'increase_inv': '<S4>:116' */
              if ((inst->bur_Sim3pCTR_B.Input3 >= inst->bur_Sim3pCTR_B.Input9) ||
                  inst->bur_Sim3pCTR_B.RelationalOperator) {
                /* Transition: '<S4>:111' */
                inst->bur_Sim3pCTR_DWork.is_inverse = Sim3pCTR_IN_steady_inv;

                /* Entry 'steady_inv': '<S4>:115' */
                inst->bur_Sim3pCTR_B.state = 0;
              }
              break;

             case Sim3pCTR_IN_steady_inv:
              /* During 'steady_inv': '<S4>:115' */
              if ((inst->bur_Sim3pCTR_B.Input3 < rtb_Add1) &&
                  (!inst->bur_Sim3pCTR_B.RelationalOperator)) {
                /* Transition: '<S4>:113' */
                inst->bur_Sim3pCTR_DWork.is_inverse = Sim3pCTR_IN_increase_inv;

                /* Entry 'increase_inv': '<S4>:116' */
                inst->bur_Sim3pCTR_B.state = 1;
              } else {
                if ((inst->bur_Sim3pCTR_B.Input3 > rtb_Add) &&
                    (!inst->bur_Sim3pCTR_B.RelationalOperator1)) {
                  /* Transition: '<S4>:114' */
                  inst->bur_Sim3pCTR_DWork.is_inverse = Sim3pCTR_IN_decrease_inv;

                  /* Entry 'decrease_inv': '<S4>:117' */
                  inst->bur_Sim3pCTR_B.state = 2;
                }
              }
              break;

             default:
              /* Transition: '<S4>:110' */
              inst->bur_Sim3pCTR_DWork.is_inverse = Sim3pCTR_IN_steady_inv;

              /* Entry 'steady_inv': '<S4>:115' */
              inst->bur_Sim3pCTR_B.state = 0;
              break;
            }
          }
          break;

         case Sim3pCTR_IN_normal:
          /* During 'normal': '<S4>:106' */
          if (inst->bur_Sim3pCTR_B.Input14 == TRUE) {
            /* Transition: '<S4>:120' */
            inst->bur_Sim3pCTR_DWork.is_normal = (uint8_T)Sim3pCTR_IN_NO_ACTIVE_CHILD;
            inst->bur_Sim3pCTR_DWork.is_enabled = Sim3pCTR_IN_inverse;

            /* Transition: '<S4>:110' */
            inst->bur_Sim3pCTR_DWork.is_inverse = Sim3pCTR_IN_steady_inv;

            /* Entry 'steady_inv': '<S4>:115' */
            inst->bur_Sim3pCTR_B.state = 0;
          } else {
            switch (inst->bur_Sim3pCTR_DWork.is_normal) {
             case Sim3pCTR_IN_decrease:
              /* During 'decrease': '<S4>:25' */
              if ((inst->bur_Sim3pCTR_B.Input3 <= inst->bur_Sim3pCTR_B.Input9) ||
                  inst->bur_Sim3pCTR_B.RelationalOperator) {
                /* Transition: '<S4>:27' */
                inst->bur_Sim3pCTR_DWork.is_normal = Sim3pCTR_IN_steady;

                /* Entry 'steady': '<S4>:11' */
                inst->bur_Sim3pCTR_B.state = 0;
              }
              break;

             case Sim3pCTR_IN_increase:
              /* During 'increase': '<S4>:24' */
              if ((inst->bur_Sim3pCTR_B.Input3 >= inst->bur_Sim3pCTR_B.Input9) ||
                  inst->bur_Sim3pCTR_B.RelationalOperator1) {
                /* Transition: '<S4>:31' */
                inst->bur_Sim3pCTR_DWork.is_normal = Sim3pCTR_IN_steady;

                /* Entry 'steady': '<S4>:11' */
                inst->bur_Sim3pCTR_B.state = 0;
              }
              break;

             case Sim3pCTR_IN_steady:
              /* During 'steady': '<S4>:11' */
              if ((inst->bur_Sim3pCTR_B.Input3 > rtb_Add) &&
                  (!inst->bur_Sim3pCTR_B.RelationalOperator)) {
                /* Transition: '<S4>:29' */
                inst->bur_Sim3pCTR_DWork.is_normal = Sim3pCTR_IN_decrease;

                /* Entry 'decrease': '<S4>:25' */
                inst->bur_Sim3pCTR_B.state = 1;
              } else {
                if ((inst->bur_Sim3pCTR_B.Input3 < rtb_Add1) &&
                    (!inst->bur_Sim3pCTR_B.RelationalOperator1)) {
                  /* Transition: '<S4>:32' */
                  inst->bur_Sim3pCTR_DWork.is_normal = Sim3pCTR_IN_increase;

                  /* Entry 'increase': '<S4>:24' */
                  inst->bur_Sim3pCTR_B.state = 2;
                }
              }
              break;

             default:
              /* Transition: '<S4>:78' */
              inst->bur_Sim3pCTR_DWork.is_normal = Sim3pCTR_IN_steady;

              /* Entry 'steady': '<S4>:11' */
              inst->bur_Sim3pCTR_B.state = 0;
              break;
            }
          }
          break;

         default:
          /* Transition: '<S4>:123' */
          inst->bur_Sim3pCTR_DWork.is_enabled = Sim3pCTR_IN_normal;

          /* Transition: '<S4>:78' */
          inst->bur_Sim3pCTR_DWork.is_normal = Sim3pCTR_IN_steady;

          /* Entry 'steady': '<S4>:11' */
          inst->bur_Sim3pCTR_B.state = 0;
          break;
        }
      }
      break;

     case Sim3pCTR_IN_manual_ramp:
      /* During 'manual_ramp': '<S4>:86' */
      if (inst->bur_Sim3pCTR_B.Input == FALSE) {
        /* Transition: '<S4>:98' */
        inst->bur_Sim3pCTR_DWork.is_manual_ramp = (uint8_T)Sim3pCTR_IN_NO_ACTIVE_CHILD;
        inst->bur_Sim3pCTR_DWork.is_c1_Sim3pCTR = Sim3pCTR_IN_disabled;

        /* Entry 'disabled': '<S4>:69' */
        inst->bur_Sim3pCTR_B.state = 0;
      } else if ((!inst->bur_Sim3pCTR_B.Input13) && (!inst->bur_Sim3pCTR_B.Input12)) {
        /* Transition: '<S4>:101' */
        inst->bur_Sim3pCTR_DWork.is_manual_ramp = (uint8_T)Sim3pCTR_IN_NO_ACTIVE_CHILD;
        inst->bur_Sim3pCTR_DWork.is_c1_Sim3pCTR = Sim3pCTR_IN_enabled;

        /* Transition: '<S4>:123' */
        inst->bur_Sim3pCTR_DWork.is_enabled = Sim3pCTR_IN_normal;

        /* Transition: '<S4>:78' */
        inst->bur_Sim3pCTR_DWork.is_normal = Sim3pCTR_IN_steady;

        /* Entry 'steady': '<S4>:11' */
        inst->bur_Sim3pCTR_B.state = 0;
      } else {
        switch (inst->bur_Sim3pCTR_DWork.is_manual_ramp) {
         case Sim3pCTR_IN_man_decrease:
          /* During 'man_decrease': '<S4>:90' */
          if ((!inst->bur_Sim3pCTR_B.Input12) || inst->bur_Sim3pCTR_B.RelationalOperator) {
            /* Transition: '<S4>:95' */
            inst->bur_Sim3pCTR_DWork.is_manual_ramp = Sim3pCTR_IN_man_steady;

            /* Entry 'man_steady': '<S4>:88' */
            inst->bur_Sim3pCTR_B.state = 0;
          }
          break;

         case Sim3pCTR_IN_man_increase:
          /* During 'man_increase': '<S4>:89' */
          if ((!inst->bur_Sim3pCTR_B.Input13) || inst->bur_Sim3pCTR_B.RelationalOperator1 ||
              inst->bur_Sim3pCTR_B.Input12) {
            /* Transition: '<S4>:92' */
            inst->bur_Sim3pCTR_DWork.is_manual_ramp = Sim3pCTR_IN_man_steady;

            /* Entry 'man_steady': '<S4>:88' */
            inst->bur_Sim3pCTR_B.state = 0;
          }
          break;

         case Sim3pCTR_IN_man_steady:
          /* During 'man_steady': '<S4>:88' */
          if (inst->bur_Sim3pCTR_B.Input12 && (!inst->bur_Sim3pCTR_B.RelationalOperator)) {
            /* Transition: '<S4>:93' */
            inst->bur_Sim3pCTR_DWork.is_manual_ramp = Sim3pCTR_IN_man_decrease;

            /* Entry 'man_decrease': '<S4>:90' */
            inst->bur_Sim3pCTR_B.state = 1;
          } else {
            if (inst->bur_Sim3pCTR_B.Input13 && (!inst->bur_Sim3pCTR_B.Input12) &&
                (!inst->bur_Sim3pCTR_B.RelationalOperator1)) {
              /* Transition: '<S4>:91' */
              inst->bur_Sim3pCTR_DWork.is_manual_ramp = Sim3pCTR_IN_man_increase;

              /* Entry 'man_increase': '<S4>:89' */
              inst->bur_Sim3pCTR_B.state = 2;
            }
          }
          break;

         default:
          /* Transition: '<S4>:87' */
          inst->bur_Sim3pCTR_DWork.is_manual_ramp = Sim3pCTR_IN_man_steady;

          /* Entry 'man_steady': '<S4>:88' */
          inst->bur_Sim3pCTR_B.state = 0;
          break;
        }
      }
      break;

     default:
      /* Transition: '<S4>:79' */
      inst->bur_Sim3pCTR_DWork.is_c1_Sim3pCTR = Sim3pCTR_IN_disabled;

      /* Entry 'disabled': '<S4>:69' */
      inst->bur_Sim3pCTR_B.state = 0;
      break;
    }
  }

  /* End of Stateflow: '<S2>/StateMachine' */

  /* Switch: '<S3>/Switch1' incorporates:
   *  Product: '<S3>/Product'
   *  Sum: '<S3>/Add'
   */
  if (inst->bur_Sim3pCTR_B.Input7) {
    rtb_Add = inst->bur_Sim3pCTR_B.Input8;
  } else {
    /* MultiPortSwitch: '<S2>/Multiport Switch' incorporates:
     *  Constant: '<S2>/Constant'
     *  Gain: '<S2>/Gain'
     */
    switch (inst->bur_Sim3pCTR_B.state) {
     case 0:
      rtb_Add = 0.0F;
      break;

     case 1:
      rtb_Add = -inst->bur_Sim3pCTR_B.Input5;
      break;

     default:
      rtb_Add = inst->bur_Sim3pCTR_B.Input4;
      break;
    }

    /* End of MultiPortSwitch: '<S2>/Multiport Switch' */
    rtb_Add = rtb_Add * inst->bur_Sim3pCTR_B.Input6 + inst->bur_Sim3pCTR_B.Switch2;
  }

  /* End of Switch: '<S3>/Switch1' */

  /* Update for UnitDelay: '<S3>/Unit Delay' */
  inst->bur_Sim3pCTR_DWork.UnitDelay_DSTATE = rtb_Add;

  /* End of Outputs for SubSystem: '<Root>/Sim3pCTR' */

  /* S-Function (bur_out): '<Root>/Output' */
  inst->Y = inst->bur_Sim3pCTR_B.Switch2;

  /* S-Function (bur_out): '<Root>/Output1' */
  inst->bY_min_limit = inst->bur_Sim3pCTR_B.RelationalOperator;

  /* S-Function (bur_out): '<Root>/Output2' */
  inst->bY_max_limit = inst->bur_Sim3pCTR_B.RelationalOperator1;

  /* S-Function (bur_out): '<Root>/Output3' */
  inst->State = inst->bur_Sim3pCTR_B.state;
}

/* Model initialize function */
void Sim3pCTR_initialize(struct Sim3pCTR* inst)
{
  /* (no initialization code required) */
}

/* Model terminate function */
void Sim3pCTR_terminate(struct Sim3pCTR* inst)
{
  /* (no terminate code required) */
}

/*======================== TOOL VERSION INFORMATION ==========================*
 * MATLAB 7.12 (R2011a)09-Mar-2011                                            *
 * Simulink 7.7 (R2011a)09-Mar-2011                                           *
 * Simulink Coder 8.0 (R2011a)09-Mar-2011                                     *
 * Embedded Coder 6.0 (R2011a)09-Mar-2011                                     *
 * Stateflow 7.7 (R2011a)09-Mar-2011                                          *
 * Simulink Fixed Point 6.5 (R2011a)09-Mar-2011                               *
 *============================================================================*/

/*======================= LICENSE IN USE INFORMATION =========================*
 * matlab                                                                     *
 * matlab_coder                                                               *
 * real-time_workshop                                                         *
 * rtw_embedded_coder                                                         *
 * simulink                                                                   *
 * stateflow                                                                  *
 *============================================================================*/
```
